# B&R Automation Studio project Y4_V3_1 (part 7)

#### Page13.st - Cyclic code
```iecst
(********************************************************************
 * COPYRIGHT --
 ********************************************************************
 * Program: Page13
 * File: Page13.st
 * Author: NickE
 * Created: January 31, 2013
 ********************************************************************
 * Implementation of program Page13
 ********************************************************************)

PROGRAM _CYCLIC

	//SETTINGS SCREEN
	Vis.P13.EnableIndex	:=	LIMIT(0,Vis.P13.EnableIndex,24)	;
	Vis.P13.Status[0]	:=	HIDE	;
	Vis.P13.Status[1]	:=	HIDE	;
	Vis.P13.Status[2]	:=	HIDE	;
	Vis.P13.Status[3]	:=	HIDE	;
	Vis.P13.Status[4]	:=	HIDE	;
	Vis.P13.Status[5]	:=	HIDE	;
	Vis.P13.Status[6]	:=	HIDE	;
	Vis.P13.Status[7]	:=	HIDE	;
	Vis.P13.Status[8]	:=	HIDE	;
	Vis.P13.Status[9]	:=	HIDE	;
	Vis.P13.Status[10]	:=	HIDE	;
	Vis.P13.Colour[1]	:=	BLUE	;
	Vis.P13.Colour[2]	:=	BLUE	;
	Vis.P13.Colour[3]	:=	BLUE	;
	Vis.P13.Colour[4]	:=	BLUE	;
	Vis.P13.Colour[5]	:=	BLUE	;
	Vis.P13.Colour[6]	:=	BLUE	;

	CASE Vis.P13.EnableIndex OF
		0:
			Vis.P13.Status[0]	:=	SHOW	;
			Vis.CalcBelt.Disp	:=	HIDE	;
		1:
			Vis.P13.Status[1]	:=	SHOW	;
			Vis.P13.Status[9]	:=	SHOW	;
			Vis.P13.Colour[1]	:=	BLUE_ACTIVE	;
		2:
			Vis.P13.Status[2]	:=	SHOW	;
			Vis.P13.Status[9]	:=	SHOW	;
			Vis.P13.Colour[2]	:=	BLUE_ACTIVE	;
			Vis.CalcBelt.Disp	:=	HIDE	;
		3:
			Vis.P13.Status[3]	:=	SHOW	;
			Vis.P13.Status[9]	:=	SHOW	;
			Vis.P13.Colour[3]	:=	BLUE_ACTIVE	;
			Vis.CalcBelt.Disp	:=	HIDE	;
		4:
			Vis.P13.Status[4]	:=	SHOW	;
			Vis.P13.Status[9]	:=	SHOW	;
			Vis.P13.Colour[4]	:=	BLUE_ACTIVE	;
			Vis.CalcBelt.Disp	:=	HIDE	;
		5:
			Vis.P13.Status[5]	:=	SHOW	;
			Vis.P13.Status[9]	:=	SHOW	;
			Vis.P13.Colour[5]	:=	BLUE_ACTIVE	;
			Vis.CalcBelt.Disp	:=	HIDE	;
		6:
			Vis.P13.Status[6]	:=	SHOW	;
			Vis.P13.Status[9]	:=	SHOW	;
			Vis.P13.Colour[6]	:=	BLUE_ACTIVE	;
			Vis.CalcBelt.Disp	:=	HIDE	;
		7:
			Vis.P13.Status[7]	:=	SHOW	;
			Vis.CalcBelt.Disp	:=	HIDE	;
		8:
			Vis.P13.Status[8]	:=	SHOW	;
			Vis.P13.Status[3]	:=	SHOW	;
			Vis.P13.Status[9]	:=	SHOW	;
			Vis.P13.Colour[3]	:=	BLUE_ACTIVE	;
			Vis.CalcBelt.Disp	:=	HIDE	;
		10:
			Vis.P13.Status[10]	:=	SHOW	;
			Vis.P13.Status[6]	:=	SHOW	;
			Vis.P13.Status[9]	:=	SHOW	;
			Vis.P13.Colour[6]	:=	BLUE_ACTIVE	;
			Vis.CalcBelt.Disp	:=	HIDE	;

	END_CASE

	//CALCULATE WHEN LAYER HAS CHANGED
	Vis.P13.Changed	:=	FALSE	;
	Vis.P13.New	:=	Vis.P13.EnableIndex	;
	IF(Vis.P13.New <> Vis.P13.Old) THEN
		Vis.P13.Changed	:=	TRUE	;
	END_IF
	IF EDGEPOS(Vis.P13.Changed) THEN
		Vis.P13Delays.EnableIndex	:=	24	;
		Vis.P13Servos.EnableIndex	:=	24	;
		Vis.P13System.EnableIndex	:=	24	;
		Vis.P13Timeouts.EnableIndex	:=	24	;
		Vis.P13Help1.EnableIndex	:=	24	;
		Vis.P13Help2.EnableIndex	:=	24	;
	END_IF
	Vis.P13.Old	:=	Vis.P13.EnableIndex	;

	//SETTINGS DELAYS SCREEN
	Vis.P13Delays.Status[0]	:=	HIDE	;
	Vis.P13Delays.Status[1]	:=	HIDE	;
	Vis.P13Delays.Status[2]	:=	HIDE	;
	Vis.P13Delays.Status[3]	:=	HIDE	;
	Vis.P13Delays.Status[4]	:=	HIDE	;
	Vis.P13Delays.Status[5]	:=	HIDE	;
	Vis.P13Delays.Status[6]	:=	HIDE	;
	Vis.P13Delays.Status[7]	:=	HIDE	;
	Vis.P13Delays.Status[8]	:=	HIDE	;
	Vis.P13Delays.Status[9]	:=	HIDE	;
	Vis.P13Delays.Status[10]	:=	HIDE	;
	Vis.P13Delays.Colour[0]	:=	BLUE	;
	Vis.P13Delays.Colour[1]	:=	BLUE	;
	Vis.P13Delays.Colour[2]	:=	BLUE	;
	Vis.P13Delays.Colour[3]	:=	BLUE	;
	Vis.P13Delays.Colour[4]	:=	BLUE	;
	Vis.P13Delays.Colour[5]	:=	BLUE	;
	Vis.P13Delays.Colour[6]	:=	BLUE	;
	Vis.P13Delays.Colour[7]	:=	BLUE	;
	Vis.P13Delays.Colour[8]	:=	BLUE	;

	CASE Vis.P13Delays.EnableIndex OF
		0..8://LayerDelay[1..9]
			Vis.P13Delays.Status[Vis.P13Delays.EnableIndex]	:=	SHOW	;
			Vis.P13Delays.Colour[Vis.P13Delays.EnableIndex]	:=	BLUE_ACTIVE	;
			Vis.P13Delays.Status[9]	:=	SHOW	;//LayerDelays
			Vis.P13.Status[1]	:=	HIDE	;//Layer2
			Vis.P13.Status[9]	:=	HIDE	;//Layers
		10:
			Vis.P13Delays.Status[10]	:=	SHOW	;
	END_CASE

	CASE Vis.P13Delays.EnableIndex OF
		0,3,4,7,8,24:
			Vis.CalcBelt.Disp	:=	HIDE	;
	END_CASE

	//CALCULATE WHEN LAYER HAS CHANGED
	Vis.P13Delays.Changed	:=	FALSE	;
	Vis.P13Delays.New	:=	Vis.P13Delays.EnableIndex	;
	IF(Vis.P13Delays.New <> Vis.P13Delays.Old) THEN
		Vis.P13Delays.Changed	:=	TRUE	;
	END_IF
	IF EDGEPOS(Vis.P13Delays.Changed) THEN
		Vis.P13Help1.EnableIndex	:=	24	;
		Vis.P13Help2.EnableIndex	:=	24	;
	END_IF
	Vis.P13Delays.Old	:=	Vis.P13Delays.EnableIndex	;

	//CALCULATOR FOR BELT DISPLAY
	IF (Vis.CalcBelt.Disp = SHOW) THEN
		IF (Vis.CalcBelt.Delay) THEN
			Vis.CalcBelt.Adjust	:= 	1 - ((Vis.CalcBelt.Unground + 300)/(Speeds.SpeedSeam/6))	;
		ELSE
			Vis.CalcBelt.Adjust	:= 	(Vis.CalcBelt.Unground + 300)/(Speeds.SpeedSeam/6);
		END_IF
		Vis.CalcBelt.New	:= 	(Vis.CalcBelt.Current + Vis.CalcBelt.Adjust)	;

		IF (Vis.CalcBelt.Unground = 0) THEN
			Vis.CalcBelt.Adjust	:= 	0	;
			Vis.CalcBelt.New	:= 	0	;
		END_IF
	END_IF

	//SETTINGS DRIVES SCREEN
	Vis.P13Drives.Status[0]	:=	HIDE	;
	Vis.P13Drives.Status[1]	:=	HIDE	;
	Vis.P13Drives.Status[2]	:=	HIDE	;
	Vis.P13Drives.Status[3]	:=	HIDE	;
	Vis.P13Drives.Status[4]	:=	HIDE	;
	Vis.P13Drives.Status[5]	:=	HIDE	;
	Vis.P13Drives.Status[6]	:=	HIDE	;
	Vis.P13Drives.Status[7]	:=	HIDE	;
	Vis.P13Drives.Status[8]	:=	HIDE	;
	Vis.P13Drives.Status[9]	:=	HIDE	;
	Vis.P13Drives.Status[10]:=	HIDE	;
	Vis.P13Drives.Status[11]:=	HIDE	;
	Vis.P13Drives.Status[12]:=	HIDE	;
	Vis.P13Drives.Status[13]:=	HIDE	;
	Vis.P13Drives.Status[14]:=	HIDE	;
	Vis.P13Drives.Status[15]:=	HIDE	;
	Vis.P13Drives.Status[20]:=	HIDE	;
	Vis.P13Drives.Status[21]:=	HIDE	;
	Vis.P13Drives.Status[22]:=	HIDE	;
	Vis.P13Drives.Colour[0]	:=	BLUE	;
	Vis.P13Drives.Colour[1]	:=	BLUE	;
	Vis.P13Drives.Colour[2]	:=	BLUE	;
	Vis.P13Drives.Colour[3]	:=	BLUE	;
	Vis.P13Drives.Colour[4]	:=	BLUE	;
	Vis.P13Drives.Colour[5]	:=	BLUE	;
	Vis.P13Drives.Colour[6]	:=	BLUE	;

	CASE Vis.P13Drives.EnableIndex OF
		0..6:
			Vis.P13Drives.Status[Vis.P13Drives.EnableIndex]	:=	SHOW	;
			Vis.P13Drives.Colour[Vis.P13Drives.EnableIndex]	:=	BLUE_ACTIVE	;
			Vis.P13Drives.Status[9]	:=	SHOW	;
			Vis.P13.Status[2]	:=	HIDE	;
			Vis.P13.Status[9]	:=	HIDE	;
			IF(Level.Level > SUPERVISOR) THEN
				Vis.P13Drives.Status[Vis.P13Drives.EnableIndex + 9]	:=	SHOW	;
			END_IF
		7:
			Vis.P13Drives.Status[7]	:=	SHOW	;
		8:
			Vis.P13Drives.Status[8]	:=	SHOW	;
	END_CASE

	CASE Vis.P13Drives.EnableIndex OF
		4:
			CASE InvPerms.CLB.Analog OF
				NO_ANALOG:
					AnalogStore.CLB.DisplayRaw := 0 ;
					AnalogStore.CLB.DisplaySpeed :=	0.0 ;
					AnalogStore.CLB.DisplayAnalog := 0.0 ;
				VOLTAGE_TYPE_1:
					AnalogStore.CLB.DisplayRaw := CLB.Input.AI1R ;
					AnalogStore.CLB.DisplaySpeed := AnalogPerm.CLB.V1.ActSpeed ;
					AnalogStore.CLB.DisplayAnalog := AnalogPerm.CLB.V1.ActAnalog ;
				CURRENT_TYPE_1:
					AnalogStore.CLB.DisplayRaw := CLB.Input.AI3R ;
					AnalogStore.CLB.DisplaySpeed := AnalogPerm.CLB.C1.ActSpeed ;
					AnalogStore.CLB.DisplayAnalog := AnalogPerm.CLB.C1.ActAnalog ;
				CURRENT_TYPE_2:
					AnalogStore.CLB.DisplayRaw := CLB.Input.AI3R ;
					AnalogStore.CLB.DisplaySpeed := AnalogPerm.CLB.C2.ActSpeed ;
					AnalogStore.CLB.DisplayAnalog := AnalogPerm.CLB.C2.ActAnalog ;
			END_CASE

			IF(AnalogStore.CLB.RecordStart) THEN
				Vis.P13Drives.Status[22]	:=	SHOW	;
			END_IF
			IF(AnalogStore.CLB.RecordConfirm) THEN
				CASE InvPerms.CLB.Analog OF
					VOLTAGE_TYPE_1:
						AnalogStore.CLB.DisplayRaw	:=	CLB.Input.AI1R	;
						AnalogPerm.CLB.V1.ActAnalog	:=	UINT_TO_REAL(AnalogStore.CLB.DisplayRaw)	;
						AnalogPerm.CLB.V1.ActSpeed	:=	AnalogStore.CLB.SpeedDisp	;
					CURRENT_TYPE_1:
						AnalogStore.CLB.DisplayRaw	:=	CLB.Input.AI3R	;
						AnalogPerm.CLB.C1.ActAnalog	:=	UINT_TO_REAL(AnalogStore.CLB.DisplayRaw)	;
						AnalogPerm.CLB.C1.ActSpeed	:=	AnalogStore.CLB.SpeedDisp	;
					CURRENT_TYPE_2:
						AnalogStore.CLB.DisplayRaw	:=	CLB.Input.AI3R	;
						AnalogPerm.CLB.C2.ActAnalog	:=	UINT_TO_REAL(AnalogStore.CLB.DisplayRaw)	;
						AnalogPerm.CLB.C2.ActSpeed	:=	AnalogStore.CLB.SpeedDisp	;
				END_CASE
				AnalogStore.CLB.RecordStart	:=	FALSE	;
				AnalogStore.CLB.RecordConfirm	:=	FALSE	;
			END_IF
		ELSE
			AnalogStore.CLB.RecordStart	:=	FALSE	;
			AnalogStore.CLB.RecordConfirm	:=	FALSE	;
	END_CASE

	//CALCULATE WHEN LAYER HAS CHANGED
	Vis.P13Drives.Changed	:=	FALSE	;
	Vis.P13Drives.New	:=	Vis.P13Drives.EnableIndex	;
	IF(Vis.P13Drives.New <> Vis.P13Drives.Old) THEN
		Vis.P13Drives.Changed	:=	TRUE	;
	END_IF
	IF EDGEPOS(Vis.P13Drives.Changed) THEN
		Vis.P13Help1.EnableIndex	:=	24	;
		Vis.P13Help2.EnableIndex	:=	24	;
	END_IF
	Vis.P13Drives.Old	:=	Vis.P13Drives.EnableIndex	;

	//SETTINGS SERVOS SCREEN
	Vis.P13Servos.Status[0]	:=	HIDE	;
	Vis.P13Servos.Status[1]	:=	HIDE	;
	Vis.P13Servos.Status[2]	:=	HIDE	;
	Vis.P13Servos.Status[3]	:=	HIDE	;
	Vis.P13Servos.Status[4]	:=	HIDE	;
	Vis.P13Servos.Status[5]	:=	HIDE	;
	Vis.P13Servos.Status[6]	:=	HIDE	;
	Vis.P13Servos.Status[7]	:=	HIDE	;
	Vis.P13Servos.Status[8]	:=	HIDE	;
	Vis.P13Servos.Status[9]	:=	HIDE	;
	Vis.P13Servos.Colour[0]	:=	BLUE	;
	Vis.P13Servos.Colour[1]	:=	BLUE	;
	Vis.P13Servos.Colour[2]	:=	BLUE	;
	Vis.P13Servos.Colour[3]	:=	BLUE	;
	Vis.P13Servos.Colour[4]	:=	BLUE	;
	Vis.P13Servos.Colour[5]	:=	BLUE	;
	Vis.P13Servos.Colour[6]	:=	BLUE	;

	CASE Vis.P13Servos.EnableIndex OF
		0..6:
			Vis.P13Servos.Status[Vis.P13Servos.EnableIndex]	:=	SHOW	;
			Vis.P13Servos.Colour[Vis.P13Servos.EnableIndex]	:=	BLUE_ACTIVE	;
			Vis.P13Servos.Status[9]	:=	SHOW	;
			Vis.P13.Status[2]	:=	HIDE	;
			Vis.P13.Status[9]	:=	HIDE	;
		7:
			Vis.P13Servos.Status[7]	:=	SHOW	;
		8:
			Vis.P13Servos.Status[8]	:=	SHOW	;
	END_CASE

	//CALCULATE WHEN LAYER HAS CHANGED
	Vis.P13Servos.Changed	:=	FALSE	;
	Vis.P13Servos.New	:=	Vis.P13Servos.EnableIndex	;
	IF(Vis.P13Servos.New <> Vis.P13Servos.Old) THEN
		Vis.P13Servos.Changed	:=	TRUE	;
	END_IF
	IF EDGEPOS(Vis.P13Servos.Changed) THEN
		Vis.P13Help1.EnableIndex	:=	24	;
		Vis.P13Help2.EnableIndex	:=	24	;
	END_IF
	Vis.P13Servos.Old	:=	Vis.P13Servos.EnableIndex	;

	//SETTINGS SYSTEM SCREEN
	Vis.P13System.Status[0]	:=	HIDE	;
	Vis.P13System.Status[1]	:=	HIDE	;
	Vis.P13System.Status[2]	:=	HIDE	;
	Vis.P13System.Status[3]	:=	HIDE	;
	Vis.P13System.Status[4]	:=	HIDE	;
	Vis.P13System.Status[5]	:=	HIDE	;
	Vis.P13System.Status[6]	:=	HIDE	;
	Vis.P13System.Status[7]	:=	HIDE	;
	Vis.P13System.Status[8]	:=	HIDE	;
	Vis.P13System.Status[9]	:=	HIDE	;
	Vis.P13System.Colour[0]	:=	BLUE	;
	Vis.P13System.Colour[1]	:=	BLUE	;
	Vis.P13System.Colour[2]	:=	BLUE	;
	Vis.P13System.Colour[3]	:=	BLUE	;
	Vis.P13System.Colour[4]	:=	BLUE	;
	Vis.P13System.Colour[5]	:=	BLUE	;
	Vis.P13System.Colour[6]	:=	BLUE	;

	CASE Vis.P13System.EnableIndex OF
		0..6:
			Vis.P13System.Status[Vis.P13System.EnableIndex]	:=	SHOW	;
			Vis.P13System.Colour[Vis.P13System.EnableIndex]	:=	BLUE_ACTIVE	;
			Vis.P13System.Status[9]	:=	SHOW	;
			Vis.P13.Status[4]	:=	HIDE	;
			Vis.P13.Status[9]	:=	HIDE	;
		7:
			Vis.P13System.Status[7]	:=	SHOW	;
		8:
			Vis.P13System.Status[8]	:=	SHOW	;
	END_CASE

	//CALCULATE WHEN LAYER HAS CHANGED
	Vis.P13System.Changed	:=	FALSE	;
	Vis.P13System.New	:=	Vis.P13System.EnableIndex	;
	IF(Vis.P13System.New <> Vis.P13System.Old) THEN
		Vis.P13System.Changed	:=	TRUE	;
	END_IF
	IF EDGEPOS(Vis.P13System.Changed) THEN
		Vis.P13Help1.EnableIndex	:=	24	;
		Vis.P13Help2.EnableIndex	:=	24	;
	END_IF
	Vis.P13System.Old	:=	Vis.P13System.EnableIndex	;

	//SETTINGS TIMEOUT SCREEN
	Vis.P13Timeouts.Status[0]	:=	HIDE	;
	Vis.P13Timeouts.Status[1]	:=	HIDE	;
	Vis.P13Timeouts.Status[2]	:=	HIDE	;
	Vis.P13Timeouts.Status[3]	:=	HIDE	;
	Vis.P13Timeouts.Status[4]	:=	HIDE	;
	Vis.P13Timeouts.Status[5]	:=	HIDE	;
	Vis.P13Timeouts.Status[6]	:=	HIDE	;
	Vis.P13Timeouts.Status[7]	:=	HIDE	;
	Vis.P13Timeouts.Status[8]	:=	HIDE	;
	Vis.P13Timeouts.Status[9]	:=	HIDE	;
	Vis.P13Timeouts.Colour[0]	:=	BLUE	;
	Vis.P13Timeouts.Colour[1]	:=	BLUE	;
	Vis.P13Timeouts.Colour[2]	:=	BLUE	;
	Vis.P13Timeouts.Colour[3]	:=	BLUE	;
	Vis.P13Timeouts.Colour[4]	:=	BLUE	;
	Vis.P13Timeouts.Colour[5]	:=	BLUE	;
	Vis.P13Timeouts.Colour[6]	:=	BLUE	;

	CASE Vis.P13Timeouts.EnableIndex OF
		0..6:
			Vis.P13Timeouts.Status[Vis.P13Timeouts.EnableIndex]	:=	SHOW	;
			Vis.P13Timeouts.Colour[Vis.P13Timeouts.EnableIndex]	:=	BLUE_ACTIVE	;
			Vis.P13Timeouts.Status[9]	:=	SHOW	;
			Vis.P13.Status[5]	:=	HIDE	;
			Vis.P13.Status[9]	:=	HIDE	;
		7:
			Vis.P13Timeouts.Status[7]	:=	SHOW	;
		8:
			Vis.P13Timeouts.Status[8]	:=	SHOW	;
	END_CASE

	//CALCULATE WHEN LAYER HAS CHANGED
	Vis.P13Timeouts.Changed	:=	FALSE	;
	Vis.P13Timeouts.New	:=	Vis.P13Timeouts.EnableIndex	;
	IF(Vis.P13Timeouts.New <> Vis.P13Timeouts.Old) THEN
		Vis.P13Timeouts.Changed	:=	TRUE	;
	END_IF
	IF EDGEPOS(Vis.P13Timeouts.Changed) THEN
		Vis.P13Help1.EnableIndex	:=	24	;
		Vis.P13Help2.EnableIndex	:=	24	;
	END_IF
	Vis.P13Timeouts.Old	:=	Vis.P13Timeouts.EnableIndex	;

	//HELP LAYERS CONTROL
	memcpy(ADR(Vis.P13Help1.Status),ADR(Vis.HideAll),SIZEOF(Vis.HideAll));
	Vis.P13Help1.Colour[0]	:=	BLUE	;
	Vis.P13Help1.Colour[1]	:=	BLUE	;
	Vis.P13Help1.Colour[2]	:=	BLUE	;
	Vis.P13Help1.Colour[3]	:=	BLUE	;
	Vis.P13Help1.Colour[4]	:=	BLUE	;
	Vis.P13Help1.Colour[5]	:=	BLUE	;
	Vis.P13Help1.Colour[6]	:=	BLUE	;
	Vis.P13Help1.Colour[7]	:=	BLUE	;
	Vis.P13Help1.Colour[8]	:=	BLUE	;
	Vis.P13Help1.Colour[9]	:=	BLUE	;

	CASE Vis.P13Help1.EnableIndex OF
		0..23:
			Vis.P13Help1.Status[Vis.P13Help1.EnableIndex]	:=	SHOW	;
		24:
			Vis.P13Help1.Index	:=	0	;
	END_CASE

	CASE Vis.P13Help1.Index OF
		0..9:
			Vis.P13Help1.Colour[Vis.P13Help1.Index]	:=	BLUE_ACTIVE	;
	END_CASE

	//HELP LAYERS CONTROL 2
	memcpy(ADR(Vis.P13Help2.Status),ADR(Vis.HideAll),SIZEOF(Vis.HideAll));
	Vis.P13Help2.Colour[0]	:=	BLUE	;
	Vis.P13Help2.Colour[1]	:=	BLUE	;
	Vis.P13Help2.Colour[2]	:=	BLUE	;
	Vis.P13Help2.Colour[3]	:=	BLUE	;
	Vis.P13Help2.Colour[4]	:=	BLUE	;
	Vis.P13Help2.Colour[5]	:=	BLUE	;
	Vis.P13Help2.Colour[6]	:=	BLUE	;
	Vis.P13Help2.Colour[7]	:=	BLUE	;
	Vis.P13Help2.Colour[8]	:=	BLUE	;
	Vis.P13Help2.Colour[9]	:=	BLUE	;
	Vis.P13Help2.Colour[10]	:=	BLUE	;

	CASE Vis.P13Help2.EnableIndex OF
		0..23:
			Vis.P13Help2.Status[Vis.P13Help2.EnableIndex]	:=	SHOW	;
		24:
			Vis.P13Help2.Index	:=	0	;
	END_CASE

	CASE Vis.P13Help2.Index OF
		0..10:
			Vis.P13Help2.Colour[Vis.P13Help2.Index]	:=	BLUE_ACTIVE	;
	END_CASE

END_PROGRAM
```

### Program Logical/VisControl/HMIControl/Page14 (IEC) - Drives screen

#### Page14.st - Cyclic code
```iecst
(********************************************************************
 * COPYRIGHT --
 ********************************************************************
 * Program: Page14
 * File: Page14.st
 * Author: NickE
 * Created: January 31, 2013
 ********************************************************************
 * Implementation of program Page14
 ********************************************************************)

PROGRAM _CYCLIC

	//DRIVES SCREEN
	memcpy(ADR(Vis.P14.Status),ADR(Vis.HideAll),SIZEOF(Vis.HideAll));
	Vis.P14.Colour[0]	:=	VIOLET	;
	Vis.P14.Colour[1]	:=	VIOLET	;
	Vis.P14.Colour[2]	:=	VIOLET	;
	Vis.P14.Colour[3]	:=	VIOLET	;
	Vis.P14.Colour[4]	:=	VIOLET	;
	Vis.P14.Colour[5]	:=	VIOLET	;
	Vis.P14.Colour[6]	:=	VIOLET	;

	CASE Vis.P14.EnableIndex OF
		0..6:
			Vis.P14.Status[Vis.P14.EnableIndex]	:=	SHOW	;
			Vis.P14.Colour[Vis.P14.EnableIndex]	:=	VIOLET_ACTIVE	;
	END_CASE

	IF (Control.Test) THEN
		Vis.P14.Status[8]	:=	SHOW	;
	END_IF

	IF(Control.Test) THEN
		Vis.P14.Status[9]	:=	SHOW	;
	END_IF

	//CALCULATE WHEN LAYER HAS CHANGED
	Vis.P14.Changed	:=	FALSE	;
	Vis.P14.New	:=	Vis.P14.EnableIndex	;
	IF(Vis.P14.New <> Vis.P14.Old) THEN
		Vis.P14.Changed	:=	TRUE	;
	END_IF
	IF EDGEPOS(Vis.P14.Changed) THEN
		Vis.P14Layer.EnableIndex	:=	24	;
		Vis.P14Status.EnableIndex	:=	24	;
		Vis.P14Help.EnableIndex		:=	24	;
		//		Vis.CalcFreq.Disp				:=	HIDE	;
	END_IF
	Vis.P14.Old	:=	Vis.P14.EnableIndex	;

	memcpy(ADR(Vis.P14Layer.Status),ADR(Vis.HideAll),SIZEOF(Vis.HideAll));

	CASE Vis.P14Layer.EnableIndex OF
		0..19:
			Vis.P14Layer.Status[Vis.P14Layer.EnableIndex]	:=	SHOW	;
//		24:
//			Vis.CalcFreq.Disp	:=	HIDE	;
	END_CASE

	IF NOT(Control.Test) THEN
		Vis.P14Layer.EnableIndex	:= 24	;
	END_IF

	memcpy(ADR(Vis.P14Status.Status),ADR(Vis.HideAll),SIZEOF(Vis.HideAll));

	CASE Vis.P14Status.EnableIndex OF
		0..19:
			Vis.P14Status.Status[Vis.P14Status.EnableIndex]	:=	SHOW	;
	END_CASE

	memcpy(ADR(Vis.P14Help.Status),ADR(Vis.HideAll),SIZEOF(Vis.HideAll));

	CASE Vis.P14Help.EnableIndex OF
		0..15:
			Vis.P14Help.Status[Vis.P14Help.EnableIndex]	:=	SHOW	;
	END_CASE

	//DISPLAY INVERTER RESET BUTTON
	FOR i := 16 TO 31 DO
		IF(SysTemp.Alarms[i])THEN
			Vis.P14.Status[23]	:=	SHOW	;
		END_IF
	END_FOR
	IF(InvReset.Auto) AND(CL1.Input.Fault) THEN
		CL1.Output.CMDD_07	:=	TRUE	;
	END_IF
	IF(InvReset.Auto) AND(CS1.Input.Fault) THEN
		CS1.Output.CMDD_07	:=	TRUE	;
	END_IF
	IF(InvReset.Auto) AND(CV1.Input.Fault) THEN
		CV1.Output.CMDD_07	:=	TRUE	;
	END_IF
	IF(InvReset.Auto) AND(CC1.Input.Fault) THEN
		CC1.Output.CMDD_07	:=	TRUE	;
	END_IF
	IF(InvReset.Auto) AND(CC2.Input.Fault) THEN
		CC2.Output.CMDD_07	:=	TRUE	;
	END_IF
	IF(InvReset.Auto) AND(CS2.Input.Fault) THEN
		CS2.Output.CMDD_07	:=	TRUE	;
	END_IF
	IF(InvReset.Auto) AND(CV2.Input.Fault) THEN
		CV2.Output.CMDD_07	:=	TRUE	;
	END_IF
	IF(InvReset.Auto) AND(CC3.Input.Fault) THEN
		CC3.Output.CMDD_07	:=	TRUE	;
	END_IF
	IF(InvReset.Auto) AND(CC4.Input.Fault) THEN
		CC4.Output.CMDD_07	:=	TRUE	;
	END_IF
	IF(InvReset.Auto) AND(CB1.Input.Fault) THEN
		CB1.Output.CMDD_07	:=	TRUE	;
	END_IF
	IF(InvReset.Auto) AND(CB2.Input.Fault) THEN
		CB2.Output.CMDD_07	:=	TRUE	;
	END_IF
	IF(InvReset.Auto) AND(CRB.Input.Fault) THEN
		CRB.Output.CMDD_07	:=	TRUE	;
	END_IF
	IF(InvReset.Auto) AND(CRE.Input.Fault) THEN
		CRE.Output.CMDD_07	:=	TRUE	;
	END_IF
	IF(InvReset.Auto) AND(CLB.Input.Fault) THEN
		CLB.Output.CMDD_07	:=	TRUE	;
	END_IF

END_PROGRAM
```

### Program Logical/VisControl/HMIControl/Page15 (IEC) - Servo screen controls

#### Page15.st - Cyclic code
```iecst
(********************************************************************
 * COPYRIGHT --
 ********************************************************************
 * Program: Page15
 * File: Page15.st
 * Author: nicke
 * Created: February 04, 2013
 ********************************************************************
 * Implementation of program Page15
 ********************************************************************)

PROGRAM _CYCLIC

	//SERVOS SCREEN
	memcpy(ADR(Vis.P15.Status),ADR(Vis.HideAll),SIZEOF(Vis.HideAll));
	Vis.P15.Colour[0]	:=	GREEN1	;
	Vis.P15.Colour[1]	:=	GREEN1	;
	Vis.P15.Colour[2]	:=	GREEN1	;
	Vis.P15.Colour[3]	:=	GREEN1	;
	Vis.P15.Colour[4]	:=	GREEN1	;
	Vis.P15.Colour[5]	:=	GREEN1	;
	Vis.P15.Colour[6]	:=	GREEN1	;

	CASE Vis.P15.EnableIndex OF
		0..6:
			Vis.P15.Status[Vis.P15.EnableIndex]	:=	SHOW	;
			Vis.P15.Colour[Vis.P15.EnableIndex]	:=	GREEN1_ACTIVE	;
	END_CASE

	IF(Control.Test) THEN
		Vis.P15.Status[8]	:=	SHOW	;
		//	ELSE
		//		Vis.P15Layer.EnableIndex	:=	24	;
	END_IF

	//CALCULATE WHEN LAYER HAS CHANGED
	Vis.P15.Changed	:=	FALSE	;
	Vis.P15.New	:=	Vis.P15.EnableIndex	;
	IF(Vis.P15.New <> Vis.P15.Old) THEN
		Vis.P15.Changed	:=	TRUE	;
	END_IF
	IF EDGEPOS(Vis.P15.Changed) THEN
		Vis.P15Layer.EnableIndex	:=	24	;
	END_IF
	Vis.P15.Old	:=	Vis.P15.EnableIndex	;

	memcpy(ADR(Vis.P15Layer.Status),ADR(Vis.HideAll),SIZEOF(Vis.HideAll));

	CASE Vis.P15Layer.EnableIndex OF
		0..15:
			Vis.P15Layer.Status[Vis.P15Layer.EnableIndex]	:=	SHOW	;
	END_CASE

	IF(Control.Test) THEN
		TestServos	:=	TRUE	;
	ELSE
		TestServos	:=	FALSE	;
		Vis.P15Layer.Status[0]	:=	HIDE	;
		Vis.P15Layer.Status[1]	:=	HIDE	;
		Vis.P15Layer.Status[2]	:=	HIDE	;
	END_IF

	Ax1.Seek2Runtime	:=	(BOOL_TO_USINT(Ax1.Block));
	Ax2.Seek2Runtime	:=	(BOOL_TO_USINT(Ax2.Block));

END_PROGRAM
```

### Program Logical/VisControl/HMIControl/Page16 (IEC) - Remote screen control

#### Page16.st - Cyclic code
```iecst
(********************************************************************
 * COPYRIGHT --
 ********************************************************************
 * Program: Page16
 * File: Page16.st
 * Author: nicke
 * Created: February 07, 2013
 ********************************************************************
 * Implementation of program Page16
 ********************************************************************)

PROGRAM _CYCLIC

	//REMOTE SCREEN
	memcpy(ADR(Vis.P16.Status),ADR(Vis.HideAll),SIZEOF(Vis.HideAll));
	Vis.P16.Colour[0]	:=	LIGHTBLUE	;
	Vis.P16.Colour[1]	:=	LIGHTBLUE	;
	Vis.P16.Colour[2]	:=	LIGHTBLUE	;
	Vis.P16.Colour[3]	:=	LIGHTBLUE	;
	Vis.P16.Colour[4]	:=	LIGHTBLUE	;
	Vis.P16.Colour[5]	:=	LIGHTBLUE	;
	Vis.P16.Colour[6]	:=	LIGHTBLUE	;
	Vis.P16.Colour[7]	:=	LIGHTBLUE	;
	Vis.P16.Colour[8]	:=	LIGHTBLUE	;
	Vis.P16.Colour[9]	:=	LIGHTBLUE	;
	Vis.P16.Colour[10]	:=	LIGHTBLUE	;

	CASE Vis.P16.EnableIndex OF
		0..7,9,10:
			Vis.P16.Status[Vis.P16.EnableIndex]	:=	SHOW	;
			Vis.P16.Colour[Vis.P16.EnableIndex]	:=	LIGHTBLUE_ACTIVE	;
	END_CASE

	IF(Control.Test) THEN
		Vis.P16.Status[8]	:=	SHOW	;
	ELSE
		Vis.P16.EnableIndex	:= LIMIT(0, Vis.P16.EnableIndex, 5);//ALTER Limit max dependent on number of IO screens, 5=6 screens ETC...
	END_IF

	//CALCULATE WHEN LAYER HAS CHANGED
	Vis.P16.Changed	:=	FALSE	;
	Vis.P16.New	:=	Vis.P16.EnableIndex	;
	IF(Vis.P16.New <> Vis.P16.Old) THEN
		Vis.P16.Changed	:=	TRUE	;
	END_IF
	IF EDGEPOS(Vis.P16.Changed) THEN
		Vis.P16Layer.EnableIndex	:=	24	;
	END_IF
	Vis.P16.Old	:=	Vis.P16.EnableIndex	;

	memcpy(ADR(Vis.P16Layer.Status),ADR(Vis.HideAll),SIZEOF(Vis.HideAll));

	CASE Vis.P16Layer.EnableIndex OF
		0..15:
			Vis.P16Layer.Status[Vis.P16Layer.EnableIndex]	:=	SHOW	;
	END_CASE

	//Declaration to enable use of variables on screen
	X2XModule	;

END_PROGRAM
```

### Program Logical/VisControl/HMIControl/Page17 (IEC) - Alarm screen control

#### Page17.st - Cyclic code
```iecst
(********************************************************************
 * COPYRIGHT -ASHTON INDUSTRIAL 2016-
 ********************************************************************
 * Program: Page17
 * File: Page17.st
 * Author: NE
 ********************************************************************)

PROGRAM _CYCLIC

	Alarm.Control := 3 ;  	//Enable Alarm Index selection
	Alarm.Group := 1 ;	// Equals alarm group index
	Alarm.Alarm := 0 ;	// Not used
	Alarm.Priority := 0 ;	// Not used

	// Convert alarm inputs to alarm array
	SysTemp.Alarms[0] := MS1Belt1.Trip ;
	SysTemp.Alarms[1] := MS2Belt2.Trip ;
	SysTemp.Alarms[2] := MS3Belt3.Trip ;
	SysTemp.Alarms[3] := MS4Belt4.Trip ;
	SysTemp.Alarms[4] := MS5Belt5.Trip ;
	SysTemp.Alarms[5] := MS6Belt6.Trip ;
	SysTemp.Alarms[6] := MS7Belt7.Trip ;
	SysTemp.Alarms[7] := MS8Belt8.Trip ;
	SysTemp.Alarms[8] := MS9Vac1.Trip ;
	SysTemp.Alarms[9] := MS10Vac2.Trip ;
	SysTemp.Alarms[10] := MS11Vac3.Trip ;
	SysTemp.Alarms[11] := MS12Vac4.Trip ;
	SysTemp.Alarms[12] := MS13Water1.Trip ;
	SysTemp.Alarms[13] := MS14Water2.Trip ;
	SysTemp.Alarms[14] := (CL1.Input.Fault) ;
	SysTemp.Alarms[15] := (CS1.Input.Fault) ;
	SysTemp.Alarms[16] := (CV1.Input.Fault) ;
	SysTemp.Alarms[17] := (CC1.Input.Fault) ;
	SysTemp.Alarms[18] := (CC2.Input.Fault) ;
	SysTemp.Alarms[19] := (CS2.Input.Fault) ;
	SysTemp.Alarms[20] := (CV2.Input.Fault) ;
	SysTemp.Alarms[21] := (CC3.Input.Fault) ;
	SysTemp.Alarms[22] := (CC4.Input.Fault) ;
	SysTemp.Alarms[23] := (CB1.Input.Fault) ;
	SysTemp.Alarms[24] := (CB2.Input.Fault) ;
	SysTemp.Alarms[25] := (CRB.Input.Fault) ;
	SysTemp.Alarms[26] := (CRE.Input.Fault) ;
	SysTemp.Alarms[27] := (CLB.Input.Fault) ;
	SysTemp.Alarms[28] ;
	SysTemp.Alarms[29] ;
	SysTemp.Alarms[30] ;
	SysTemp.Alarms[31] ;
	SysTemp.Alarms[32] ;
	SysTemp.Alarms[33] ;
	SysTemp.Alarms[39] := Ax1.Error AND(Control.Achieved1) ;
	SysTemp.Alarms[40] := Ax2.Error AND(Control.Achieved1) ;
	SysTemp.Alarms[41] := NOT(Servo1POT.In) ;
	SysTemp.Alarms[42] := NOT(Servo1NOT.In) ;
	SysTemp.Alarms[43] := NOT(Servo2POT.In) ;
	SysTemp.Alarms[44] := NOT(Servo2NOT.In) ;
	SysTemp.Alarms[50] := (X2XModule[5].Fuse) ;
	SysTemp.Alarms[51] := (X2XModule[6].Fuse) ;
	SysTemp.Alarms[52] := (X2XModule[7].Fuse) ;

	SysTemp.Alarm := FALSE ;
	FOR i := 0 TO 80 DO
		IF(SysTemp.Alarms[i]) THEN
			SysTemp.Alarm := TRUE ;
			EXIT ;
		END_IF
	END_FOR

END_PROGRAM
```

### Program Logical/VisControl/HMIControl/Page18 (IEC) - Warning screen control

#### Page18.st - Cyclic code
```iecst
(********************************************************************
 * COPYRIGHT --
 ********************************************************************
 * Program: Page18
 * File: Page18.st
 * Author: nicke
 * Created: April 30, 2013
 ********************************************************************
 * Implementation of program Page18
 ********************************************************************)

PROGRAM _CYCLIC

(* Section to control pop up warnings for flip arms *)
(*Seamer 1 Down *)
	Vis.FlipDisp1.Runtime1	:=	HIDE	;
	Vis.FlipDisp1.Runtime2	:=	HIDE	;
	Vis.FlipDisp1.Runtime3	:=	HIDE	;
	Vis.FlipDisp1.Runtime4	:=	HIDE	;

	IF ((Ax1.Active) OR NOT(Ax1.OriginSet)) AND NOT(Ax1.Block) AND(Control.Achieved1) THEN
		Vis.FlipDisp1.Runtime1	:=	SHOW	;
		Vis.FlipDisp1.TextIndex1	:=	BOOL_TO_USINT(NOT(S100Reed.In))	;
		Vis.FlipDisp1.TextIndex2	:=	BOOL_TO_USINT(NOT(S102Reed.In))	;
		Vis.FlipDisp1.TextIndex3	:=	BOOL_TO_USINT(NOT(S104Reed.In))	;
		Vis.FlipDisp1.TextIndex4	:=	BOOL_TO_USINT(NOT(S106Reed.In))	;
		Vis.FlipDisp1.TextIndex5	:=	BOOL_TO_USINT(NOT(S108Reed.In))	;
		Vis.FlipDisp1.TextIndex6	:=	BOOL_TO_USINT(NOT(S110Reed.In))	;
		Vis.FlipDisp1.TextIndex7	:=	BOOL_TO_USINT(NOT(S112Reed.In))	;
		Vis.FlipDisp1.TextIndex8	:=	BOOL_TO_USINT(NOT(S114Reed.In))	;
		Vis.FlipDisp1.TextIndex9	:=	BOOL_TO_USINT(NOT(S116Reed.In))	;
		Vis.FlipDisp1.TextIndex10	:=	BOOL_TO_USINT(NOT(S118Reed.In))	;
		CASE Perms.FLIPARMS1 OF
			3:
				Vis.FlipDisp1.Runtime2		:=	SHOW	;
			4:
				Vis.FlipDisp1.Runtime2		:=	SHOW	;
				Vis.FlipDisp1.Runtime3		:=	SHOW	;
			5:
				Vis.FlipDisp1.Runtime2		:=	SHOW	;
				Vis.FlipDisp1.Runtime3		:=	SHOW	;
				Vis.FlipDisp1.Runtime4		:=	SHOW	;
		END_CASE
	END_IF

	(* Seamer 1 Up *)
	Vis.FlipDisp1.Runtime5	:= HIDE	;
	Vis.FlipDisp1.Runtime6	:= HIDE	;
	Vis.FlipDisp1.Runtime7	:= HIDE	;
	Vis.FlipDisp1.Runtime8	:= HIDE	;
	Vis.FlipDisp1.Runtime9	:= HIDE	;
	Vis.FlipDisp1.TextIndex11	:=	BOOL_TO_USINT(NOT(S101Reed.In))	;
	Vis.FlipDisp1.TextIndex12	:=	BOOL_TO_USINT(NOT(S103Reed.In))	;
	Vis.FlipDisp1.TextIndex13	:=	BOOL_TO_USINT(NOT(S105Reed.In))	;
	Vis.FlipDisp1.TextIndex14	:=	BOOL_TO_USINT(NOT(S107Reed.In))	;
	Vis.FlipDisp1.TextIndex15	:=	BOOL_TO_USINT(NOT(S109Reed.In))	;
	Vis.FlipDisp1.TextIndex16	:=	BOOL_TO_USINT(NOT(S111Reed.In))	;
	Vis.FlipDisp1.TextIndex17	:=	BOOL_TO_USINT(NOT(S113Reed.In))	;
	Vis.FlipDisp1.TextIndex18	:=	BOOL_TO_USINT(NOT(S115Reed.In))	;
	Vis.FlipDisp1.TextIndex19	:=	BOOL_TO_USINT(NOT(S117Reed.In))	;
	Vis.FlipDisp1.TextIndex20	:=	BOOL_TO_USINT(NOT(S119Reed.In))	;
	CASE ArmsTemp1.CheckRaised OF
		0:	(* No arms up *)
		1:	(* 1 arm up *)
			Vis.FlipDisp1.Runtime5	:= SHOW	;
		2:	(* 2 arms up *)
			Vis.FlipDisp1.Runtime5	:= SHOW	;
			Vis.FlipDisp1.Runtime6	:= SHOW	;
		3:  (* 3 arms up *)
			Vis.FlipDisp1.Runtime5	:= SHOW	;
			Vis.FlipDisp1.Runtime6	:= SHOW	;
			Vis.FlipDisp1.Runtime7	:= SHOW	;
		4:	(* 4 arms up *)
			Vis.FlipDisp1.Runtime5	:= SHOW	;
			Vis.FlipDisp1.Runtime6	:= SHOW	;
			Vis.FlipDisp1.Runtime7	:= SHOW	;
			Vis.FlipDisp1.Runtime8	:= SHOW	;
		5:	(* 5 arms up *)
			Vis.FlipDisp1.Runtime5	:= SHOW	;
			Vis.FlipDisp1.Runtime6	:= SHOW	;
			Vis.FlipDisp1.Runtime7	:= SHOW	;
			Vis.FlipDisp1.Runtime8	:= SHOW	;
			Vis.FlipDisp1.Runtime9	:= SHOW	;
	END_CASE

	(* Seamer 2 Down *)
	Vis.FlipDisp2.Runtime1	:=	HIDE	;
	Vis.FlipDisp2.Runtime2	:=	HIDE	;
	Vis.FlipDisp2.Runtime3	:=	HIDE	;
	Vis.FlipDisp2.Runtime4	:=	HIDE	;

	IF ((Ax2.Active) OR NOT(Ax2.OriginSet)) AND NOT(Ax2.Block) AND(Control.Achieved1) THEN
		Vis.FlipDisp2.Runtime1	:=	SHOW	;
		Vis.FlipDisp2.TextIndex1	:=	BOOL_TO_USINT(NOT(S120Reed.In))	;
		Vis.FlipDisp2.TextIndex2	:=	BOOL_TO_USINT(NOT(S122Reed.In))	;
		Vis.FlipDisp2.TextIndex3	:=	BOOL_TO_USINT(NOT(S124Reed.In))	;
		Vis.FlipDisp2.TextIndex4	:=	BOOL_TO_USINT(NOT(S126Reed.In))	;
		Vis.FlipDisp2.TextIndex5	:=	BOOL_TO_USINT(NOT(S128Reed.In))	;
		Vis.FlipDisp2.TextIndex6	:=	BOOL_TO_USINT(NOT(S130Reed.In))	;
		Vis.FlipDisp2.TextIndex7	:=	BOOL_TO_USINT(NOT(S132Reed.In))	;
		Vis.FlipDisp2.TextIndex8	:=	BOOL_TO_USINT(NOT(S134Reed.In))	;
		Vis.FlipDisp2.TextIndex9	:=	BOOL_TO_USINT(NOT(S136Reed.In))	;
		Vis.FlipDisp2.TextIndex10	:=	BOOL_TO_USINT(NOT(S138Reed.In))	;
		CASE Perms.FLIPARMS2 OF
			3:
				Vis.FlipDisp2.Runtime2	:=	SHOW	;
			4:
				Vis.FlipDisp2.Runtime2	:=	SHOW	;
				Vis.FlipDisp2.Runtime3	:=	SHOW	;
			5:
				Vis.FlipDisp2.Runtime2	:=	SHOW	;
				Vis.FlipDisp2.Runtime3	:=	SHOW	;
				Vis.FlipDisp2.Runtime4	:=	SHOW	;
		END_CASE
	END_IF

	(* Seamer 2 Up *)
	Vis.FlipDisp2.Runtime5	:= HIDE	;
	Vis.FlipDisp2.Runtime6	:= HIDE	;
	Vis.FlipDisp2.Runtime7	:= HIDE	;
	Vis.FlipDisp2.Runtime8	:= HIDE	;
	Vis.FlipDisp2.Runtime9	:= HIDE	;
	Vis.FlipDisp2.TextIndex11	:=	BOOL_TO_USINT(NOT(S121Reed.In))	;
	Vis.FlipDisp2.TextIndex12	:=	BOOL_TO_USINT(NOT(S123Reed.In))	;
	Vis.FlipDisp2.TextIndex13	:=	BOOL_TO_USINT(NOT(S125Reed.In))	;
	Vis.FlipDisp2.TextIndex14	:=	BOOL_TO_USINT(NOT(S127Reed.In))	;
	Vis.FlipDisp2.TextIndex15	:=	BOOL_TO_USINT(NOT(S129Reed.In))	;
	Vis.FlipDisp2.TextIndex16	:=	BOOL_TO_USINT(NOT(S131Reed.In))	;
	Vis.FlipDisp2.TextIndex17	:=	BOOL_TO_USINT(NOT(S133Reed.In))	;
	Vis.FlipDisp2.TextIndex18	:=	BOOL_TO_USINT(NOT(S135Reed.In))	;
	Vis.FlipDisp2.TextIndex19	:=	BOOL_TO_USINT(NOT(S137Reed.In))	;
	Vis.FlipDisp2.TextIndex20	:=	BOOL_TO_USINT(NOT(S139Reed.In))	;
	CASE ArmsTemp2.CheckRaised OF
		0:	(* No arms up *)
		1:	(* 1 arm up *)
			Vis.FlipDisp2.Runtime5	:= SHOW	;
			Vis.FlipDisp2.Runtime6	:= SHOW	;
		2:	(* 2 arms up *)
			Vis.FlipDisp2.Runtime5	:= SHOW	;
			Vis.FlipDisp2.Runtime6	:= SHOW	;
			Vis.FlipDisp2.Runtime7	:= SHOW	;
		3:  (* 3 arms up *)
			Vis.FlipDisp2.Runtime5	:= SHOW	;
			Vis.FlipDisp2.Runtime6	:= SHOW	;
			Vis.FlipDisp2.Runtime7	:= SHOW	;
			Vis.FlipDisp2.Runtime8	:= SHOW	;
		4:	(* 4 arms up *)
			Vis.FlipDisp2.Runtime5	:= SHOW	;
			Vis.FlipDisp2.Runtime6	:= SHOW	;
			Vis.FlipDisp2.Runtime7	:= SHOW	;
			Vis.FlipDisp2.Runtime8	:= SHOW	;
			Vis.FlipDisp2.Runtime9	:= SHOW	;
	END_CASE

	//FILTER TO SHOW WARNINGS
	Warning.Control := 3 ; 	//Enable Alarm Index selection *)
	Warning.Group := 3 ;
	Warning.Alarm := 0 ;
	Warning.Priority := 0 ;

	Warn.Timeout[0] := Track001.TimeoutOUT ;
	Warn.Timeout[1] := Track002.TimeoutOUT ;
	Warn.Timeout[2] := Track003.TimeoutOUT ;
	Warn.Timeout[3] := Track101.TimeoutOUT ;
	Warn.Timeout[4] := Track102.TimeoutOUT ;
	Warn.Timeout[5] := Track104.TimeoutOUT ;
	Warn.Timeout[6] := Track106.TimeoutOUT ;
	Warn.Timeout[7] := Track111.TimeoutOUT ;
	Warn.Timeout[8] := Track112.TimeoutOUT ;
	Warn.Timeout[9] := Track113.TimeoutOUT ;
	Warn.Timeout[10] := Track201.TimeoutOUT ;
	Warn.Timeout[11] := Track202.TimeoutOUT ;
	Warn.Timeout[12] := Track204.TimeoutOUT ;
	Warn.Timeout[13] := Track207.TimeoutOUT ;
	Warn.Timeout[14] := Track301.TimeoutOUT ;
	Warn.Timeout[15] := Track401.TimeoutOUT ;
	Warn.Timeout[16] := Track412.TimeoutOUT ;
	Warn.Timeout[17] := Track413.TimeoutOUT ;
	Warn.Timeout[18] := Track414.TimeoutOUT ;
	Warn.Timeout[19] := Track503.TimeoutOUT ;
	Warn.Timeout[20] := Track504.TimeoutOUT ;
	Warn.Timeout[21] := Track506.TimeoutOUT ;
	Warn.Timeout[22] := Track602.TimeoutOUT ;
	Warn.Timeout[23] := Track801.TimeoutOUT ;
	Warn.Timeout[24] := Track803.TimeoutOUT ;
	Warn.Timeout[25] := Track804.TimeoutOUT ;
	Warn.Timeout[26] := Track805.TimeoutOUT ;
	Warn.Timeout[27] := Track811.TimeoutOUT ;
	Warn.Timeout[28] := Track821.TimeoutOUT ;
	Warn.Timeout[29] := Track512.TimeoutOUT ;

	FOR i:= 0 TO USINT_TO_INT(Warn.iMax) DO
		IF EDGEPOS(Warn.Timeout[i]) THEN
			Warn.Acks[i] := TRUE ;
		END_IF
	END_FOR

	FOR i:= 0 TO USINT_TO_INT(Warn.iMax) DO
		IF NOT(Warn.Timeout[i]) THEN
			Warn.Acks[i] := FALSE ;
		END_IF
	END_FOR

	//SET WARNING BIT ACTIVE WHEN TIMEOUT OCCURS
	FOR Warn.i:= 0 TO Warn.iMax DO
		IF Warn.Timeout[Warn.i] = TRUE THEN
			SysTemp.Warning :=  TRUE ;
			Warn.Button := SHOW ;
			EXIT;
		ELSE
			SysTemp.Warning := FALSE ;
			Warn.Button := HIDE ;
		END_IF
	END_FOR

	//Apply Warn.Block if EMO.Latch* are on
	IF EDGEPOS(EMO.Latch1) AND NOT(Warn.Block) THEN
		Warn.Block := TRUE ;
		Warn.BlockTemp := TRUE ;
	END_IF
	IF EDGEPOS(EMO.Latch2) AND NOT(Warn.Block) THEN
		Warn.Block := TRUE ;
		Warn.BlockTemp := TRUE ;
	END_IF

	IF EDGENEG(EMO.Latch1) AND NOT(EMO.Latch2) AND(Warn.BlockTemp) THEN
		Warn.Block := FALSE ;
		Warn.BlockTemp := FALSE ;
	END_IF
	IF EDGENEG(EMO.Latch2) AND NOT(EMO.Latch1) AND(Warn.BlockTemp) THEN
		Warn.Block := FALSE ;
		Warn.BlockTemp := FALSE ;
	END_IF

	//RESET ACK BITS IF TIMEOUT DISABLED
	IF(Warn.Block) THEN
		FOR Warn.Warningi:= 0 TO Warn.iMax DO
			Warn.Acks[Warn.Warningi]:= FALSE;
		END_FOR
	END_IF

	Warn.AckDisp	:= 	HIDE	;
	IF(SysTemp.Warning) THEN
		FOR Warn.Warningi:= 0 TO Warn.iMax DO
			IF (Warn.Acks[Warn.Warningi] = TRUE) THEN
				Warn.AckDisp	:= 	SHOW	;
				EXIT;
			ELSE
				Warn.AckDisp	:= 	HIDE	;
			END_IF
		END_FOR
	END_IF

	IF EDGEPOS(Warn.Ack) THEN
		Warn.Acks[Warn.Warningi]	:=	0	;
	END_IF

	//EVENTS
	SysTemp.Events[0] := Control.Start ;
	SysTemp.Events[1] := Control.Stop ;
	SysTemp.Events[2] := Control.EStop1 AND Control.Empty ;
	SysTemp.Events[3] := Control.EStop1 AND NOT Control.Empty ;
	SysTemp.Events[4] := SeamersII.Enable[1] ;
	SysTemp.Events[5] := SeamersII.Enable[2] ;
	SysTemp.Events[8] := SeamersII.AutoStart[0] ;
	SysTemp.Events[9] := SeamersII.AutoStart[1] ;
	SysTemp.Events[10] := SeamersII.AutoStart[2] ;
	SysTemp.Events[13] := Control.Achieved1 ;
	SysTemp.Events[14] := Control.Achieved2 ;
	SysTemp.Events[15] := Reset.Count ;
	SysTemp.Events[16] := Pause.Active ;

END_PROGRAM
```

### Program Logical/VisControl/HMIControl/Page20 (IEC) - Ashton tech screen control

#### Page20.st - Cyclic code
```iecst
(********************************************************************
 * COPYRIGHT --
 ********************************************************************
 * Program: P20
 * File: P20.st
 * Author: nicke
 * Created: February 08, 2013
 ********************************************************************
 * Implementation of program P20
 ********************************************************************)

PROGRAM _CYCLIC

	//ASHTON TECH SCREEN
	memcpy(ADR(Vis.P20.Status),ADR(Vis.HideAll),SIZEOF(Vis.HideAll));

	CASE Vis.P20.EnableIndex OF
		0..7:
			Vis.P20.Status[Vis.P20.EnableIndex]	:=	SHOW	;
	END_CASE

END_PROGRAM
```

### Program Logical/VisControl/HMIControl/ESRecover (IEC) - EStop Recovery Program

#### ESRecover.st - Cyclic code
```iecst
(********************************************************************
 * COPYRIGHT --
 ********************************************************************
 * Program: ESRecover
 * File: ESRecover.st
 * Author: NE
 ********************************************************************)

PROGRAM _CYCLIC

    //SET ESCLEAR BIT IF GLASS PRESENT AT ESTOP
	Control.ESClear := EMO.Recovery ;

	//DELAY SEAMING CONVEYORS RESTART AFTER ESTOP UNTIL GRINDING BELTS ALLOWED TO POSITION
	IF EDGENEG(Control.ESClear) THEN
		EMO.Latch1 := TRUE ;
		EMO.Latch2 := TRUE ;
	END_IF

	PresetSys.ESRestart[1] := LIMIT(10, PresetSys.ESRestart[1], 700) ;
	EMO.LatchTON1.IN := (EMO.Latch1) AND (SeamersII.DoneOUT[1]) ;
	EMO.LatchTON1.PT := PresetSys.ESRestart[1] ;
	EMO.LatchTON1 ();
	IF(EMO.LatchTON1.Q) THEN
		EMO.Latch1 := FALSE ;
	END_IF

	PresetSys.ESRestart[2] := LIMIT(10, PresetSys.ESRestart[2], 700) ;
	EMO.LatchTON2.IN := (EMO.Latch2) AND (SeamersII.DoneOUT[2]) ;
	EMO.LatchTON2.PT := PresetSys.ESRestart[2] ;
	EMO.LatchTON2 ();
	IF(EMO.LatchTON2.Q) THEN
		EMO.Latch2 := FALSE ;
	END_IF

	//AT ESTOP LATCH BIT TO ALLOW FOR MOVEMENT OF GLASS ON CONVEYORS AND PALLETS
	IF EDGEPOS(Control.EStop1) THEN
		EMO.StartLatch := TRUE ;
	END_IF

	EMO.Start.IN := EMO.StartLatch ;
	EMO.Start.PT := T#2s ;
	EMO.Start ();

	IF EDGEPOS(EMO.Start.Q) THEN
		EMO.StartLatch := FALSE ;
	END_IF

	//RESET ESCONFIRM BIT
	IF EDGEPOS(Control.EStop1) AND (Control.ESClear) OR EDGENEG(Control.ESClear) THEN
		EMO.Confirm[4] := FALSE ;
	END_IF

	//SWITCH TO EMO RECOVERY SCREEN IF ANY GLASS PRESENT
	IF EDGEPOS(Control.EStop1) AND NOT(Control.Empty) THEN
		Vis.P11.EnableIndex := 20 ;
		Vis.Page.New := P11_MIMIC ;
	END_IF

	//ESTOP RECOVERY SCREENS ACTIVE
	IF (Vis.P11.EnableIndex >= 20) AND (Vis.P11.EnableIndex <= 22) THEN
		EMO.Recovery := TRUE ;
	ELSE
		EMO.Recovery := FALSE ;
		Vis.EMO.Disp[0] := HIDE ;
		Vis.EMO.Disp[1] := HIDE ;
		Vis.EMO.Disp[2] := HIDE ;
		Vis.EMO.Disp[3] := HIDE ;
		Vis.EMO.Confirm[0] := FALSE ;
		Vis.EMO.Confirm[1] := FALSE ;
		Vis.EMO.Confirm[2] := FALSE ;
		Vis.EMO.Confirm[3] := FALSE ;
		Vis.EMO.Confirm[4] := FALSE ;
		Tracking00.Cleared := FALSE ;
		Tracking90.Cleared := FALSE ;
		Tracking01.Cleared := FALSE ;
		Tracking10.Cleared := FALSE ;
		Tracking91.Cleared := FALSE ;
		Tracking11.Cleared := FALSE ;
		Tracking20.Cleared := FALSE ;
		Tracking92.Cleared := FALSE ;
		Tracking30.Cleared := FALSE ;
		Tracking93.Cleared := FALSE ;
		Tracking40.Cleared := FALSE ;
		Tracking41.Cleared := FALSE ;
		Tracking50.Cleared := FALSE ;
		Tracking60.Cleared := FALSE ;
		Tracking70.Cleared := FALSE ;
		Tracking80.Cleared := FALSE ;
		Tracking81.Cleared := FALSE ;
		Tracking82.Cleared := FALSE ;
		Tracking51.Cleared := FALSE ;
	END_IF

	//RESET ALL BITS IF ESTOP PRESSED WHILE ON ESTOPSCREENS
	IF EDGEPOS(Control.EStop1) AND (EMO.Recovery) THEN
		Vis.EMO.Disp[0] := HIDE ;
		Vis.EMO.Disp[1] := HIDE ;
		Vis.EMO.Disp[2] := HIDE ;
		Vis.EMO.Disp[3] := HIDE ;
		Vis.EMO.Confirm[0] := FALSE ;
		Vis.EMO.Confirm[1] := FALSE ;
		Vis.EMO.Confirm[2] := FALSE ;
		Vis.EMO.Confirm[3] := FALSE ;
		Vis.EMO.Confirm[4] := FALSE ;
		Tracking00.Cleared := FALSE ;
		Tracking90.Cleared := FALSE ;
		Tracking01.Cleared := FALSE ;
		Tracking10.Cleared := FALSE ;
		Tracking91.Cleared := FALSE ;
		Tracking11.Cleared := FALSE ;
		Tracking20.Cleared := FALSE ;
		Tracking92.Cleared := FALSE ;
		Tracking30.Cleared := FALSE ;
		Tracking93.Cleared := FALSE ;
		Tracking40.Cleared := FALSE ;
		Tracking41.Cleared := FALSE ;
		Tracking50.Cleared := FALSE ;
		Tracking60.Cleared := FALSE ;
		Tracking70.Cleared := FALSE ;
		Tracking80.Cleared := FALSE ;
		Tracking81.Cleared := FALSE ;
		Tracking82.Cleared := FALSE ;
		Tracking51.Cleared := FALSE ;
	END_IF

	//ESTOP RECOVERY SCREEN CONFIRMATION AND CONTROLS
	CASE Vis.P11.EnableIndex OF
		//ESTOP SCREENS
		20:
			IF (Vis.EMO.Confirm[0]) THEN
				Vis.EMO.Disp[0] := SHOW ;
			END_IF
			IF (Vis.EMO.Confirm[1]) THEN
				Vis.EMO.Disp[1] := SHOW ;
			END_IF
			IF (Vis.EMO.Confirm[1]) AND (Control.Achieved1) THEN
				Vis.EMO.Disp[2] := SHOW;
			END_IF
		21:
			Vis.EMO.Disp[4] := SHOW ;
			IF (Vis.EMO.Confirm[2]) THEN
				Vis.EMO.Disp[3] := SHOW ;
				Vis.P11.EnableIndex := 22 ;
				Vis.EMO.Disp[4] := HIDE ;
				Vis.EMO.Confirm[4] := TRUE ;
			END_IF

			IF (Vis.EMO.Confirm[3]) THEN
				Tracking00.Cleared := FALSE ;
				Tracking90.Cleared := FALSE ;
				Tracking01.Cleared := FALSE ;
				Tracking10.Cleared := FALSE ;
				Tracking91.Cleared := FALSE ;
				Tracking11.Cleared := FALSE ;
				Tracking20.Cleared := FALSE ;
				Tracking92.Cleared := FALSE ;
				Tracking30.Cleared := FALSE ;
				Tracking93.Cleared := FALSE ;
				Tracking40.Cleared := FALSE ;
				Tracking41.Cleared := FALSE ;
				Tracking50.Cleared := FALSE ;
				Tracking60.Cleared := FALSE ;
				Tracking70.Cleared := FALSE ;
				Tracking80.Cleared := FALSE ;
				Tracking81.Cleared := FALSE ;
				Tracking82.Cleared := FALSE ;
				Tracking51.Cleared := FALSE ;
				Vis.EMO.Confirm[3] := FALSE ;
			END_IF
			//USE BITS SET FROM SCREEN TO CLEAR TRACKING DATA OF REMOVED PIECES
			Tracking00.ResES := FALSE ;
			Tracking90.ResES := FALSE ;
			Tracking01.ResES := FALSE ;
			Tracking10.ResES := FALSE ;
			Tracking91.ResES := FALSE ;
			Tracking11.ResES := FALSE ;
			Tracking20.ResES := FALSE ;
			Tracking92.ResES := FALSE ;
			Tracking30.ResES := FALSE ;
			Tracking93.ResES := FALSE ;
			Tracking40.ResES := FALSE ;
			Tracking41.ResES := FALSE ;
			Tracking50.ResES := FALSE ;
			Tracking60.ResES := FALSE ;
			Tracking70.ResES := FALSE ;
			Tracking80.ResES := FALSE ;
			Tracking81.ResES := FALSE ;
			Tracking82.ResES := FALSE ;
			Tracking51.ResES := FALSE ;
			IF EDGEPOS(Vis.EMO.Confirm[4]) THEN
				IF(Tracking00.Cleared) THEN
					Tracking00.ResES := TRUE ;
				END_IF
				IF(Tracking90.Cleared) THEN
					Tracking90.ResES := TRUE ;
				END_IF
				IF(Tracking01.Cleared) THEN
					Tracking01.ResES := TRUE ;
				END_IF
				IF(Tracking10.Cleared) THEN
					Tracking10.ResES := TRUE ;
				END_IF
				IF(Tracking91.Cleared) THEN
					Tracking91.ResES := TRUE ;
				END_IF
				IF(Tracking11.Cleared) THEN
					Tracking11.ResES := TRUE ;
				END_IF
				IF(Tracking20.Cleared) THEN
					Tracking20.ResES := TRUE ;
				END_IF
				IF(Tracking92.Cleared) THEN
					Tracking92.ResES := TRUE ;
				END_IF
				IF(Tracking30.Cleared) THEN
					Tracking30.ResES := TRUE ;
				END_IF
				IF(Tracking93.Cleared) THEN
					Tracking93.ResES := TRUE ;
				END_IF
				IF(Tracking40.Cleared) THEN
					Tracking40.ResES := TRUE ;
				END_IF
				IF(Tracking41.Cleared) THEN
					Tracking41.ResES := TRUE ;
				END_IF
				IF(Tracking50.Cleared) THEN
					Tracking50.ResES := TRUE ;
				END_IF
				IF(Tracking60.Cleared) THEN
					Tracking60.ResES := TRUE ;
				END_IF
				IF(Tracking70.Cleared) THEN
					Tracking70.ResES := TRUE ;
				END_IF
				IF(Tracking80.Cleared) THEN
					Tracking80.ResES := TRUE ;
				END_IF
				IF(Tracking81.Cleared) THEN
					Tracking81.ResES := TRUE ;
				END_IF
				IF(Tracking82.Cleared) THEN
					Tracking82.ResES := TRUE ;
				END_IF
				IF(Tracking51.Cleared) THEN
					Tracking51.ResES := TRUE ;
				END_IF

			END_IF

		22:
			//USE BITS SET FROM SCREEN TO CLEAR TRACKING DATA OF REMOVED PIECES
			Tracking00.ResES := FALSE ;
			Tracking90.ResES := FALSE ;
			Tracking01.ResES := FALSE ;
			Tracking10.ResES := FALSE ;
			Tracking91.ResES := FALSE ;
			Tracking11.ResES := FALSE ;
			Tracking20.ResES := FALSE ;
			Tracking92.ResES := FALSE ;
			Tracking30.ResES := FALSE ;
			Tracking93.ResES := FALSE ;
			Tracking40.ResES := FALSE ;
			Tracking41.ResES := FALSE ;
			Tracking50.ResES := FALSE ;
			Tracking60.ResES := FALSE ;
			Tracking70.ResES := FALSE ;
			Tracking80.ResES := FALSE ;
			Tracking81.ResES := FALSE ;
			Tracking82.ResES := FALSE ;
			Tracking51.ResES := FALSE ;
			Tracking00.Cleared := FALSE ;
			Tracking90.Cleared := FALSE ;
			Tracking01.Cleared := FALSE ;
			Tracking10.Cleared := FALSE ;
			Tracking91.Cleared := FALSE ;
			Tracking11.Cleared := FALSE ;
			Tracking20.Cleared := FALSE ;
			Tracking92.Cleared := FALSE ;
			Tracking30.Cleared := FALSE ;
			Tracking93.Cleared := FALSE ;
			Tracking40.Cleared := FALSE ;
			Tracking41.Cleared := FALSE ;
			Tracking50.Cleared := FALSE ;
			Tracking60.Cleared := FALSE ;
			Tracking70.Cleared := FALSE ;
			Tracking80.Cleared := FALSE ;
			Tracking81.Cleared := FALSE ;
			Tracking82.Cleared := FALSE ;
			Tracking51.Cleared := FALSE ;

	END_CASE

END_PROGRAM
```

### Program Logical/VisControl/HMIControl/Simulation (IEC) - Simulation control

#### Simulation.st - Cyclic code
```iecst
(********************************************************************
 * COPYRIGHT --
 ********************************************************************
 * Program: Simulation
 * File: Simulation.st
 * Author: NickE
 * Created: January 24, 2013
 ********************************************************************
 * Implementation of program Simulation
 ********************************************************************)

PROGRAM _INIT

	Control.EStop1 := TRUE ;
	Control.EStop2 := TRUE ;
	Simulation.Disp := SHOW ;
	Simulation.On := TRUE ;
	S100Reed.In := TRUE ;
	S102Reed.In := TRUE ;
	S104Reed.In := TRUE ;
	S106Reed.In := TRUE ;
	S108Reed.In := TRUE ;
	S110Reed.In := TRUE ;
	S112Reed.In := TRUE ;
	S114Reed.In := TRUE ;
	S120Reed.In := TRUE ;
	S122Reed.In := TRUE ;
	S124Reed.In := TRUE ;
	S126Reed.In := TRUE ;
	WashRun.In := TRUE ;
	CLB.Input.ETAD_02	:=	TRUE	;
	CRB.Input.ETAD_02	:=	TRUE	;

END_PROGRAM

PROGRAM _CYCLIC

	Ax1.OriginSet	:=	Control.Achieved1	;
	Ax1.Error		:=	FALSE				;
	Servo1POT.In	:= 	TRUE				;
	Servo1NOT.In	:=	TRUE				;
	Ax2.OriginSet	:=	Control.Achieved1	;
	Ax2.Error		:=	FALSE				;
	Servo2POT.In	:=	TRUE				;
	Servo2NOT.In	:=	TRUE				;

	IF EDGEPOS(Control.EStop2) THEN
		Control.EStop1	:=	TRUE	;
	END_IF

	IF NOT(TestAuto.In) THEN
		S30Reed.In	:= 	NOT(Sol30Pal1.Auto)	;
		S31Reed.In	:=	(Sol30Pal1.Auto)	;
		S32Reed.In	:= 	NOT(Sol31Pal2.Auto)	;
		S33Reed.In	:=	(Sol31Pal2.Auto)	;
		S34Reed.In	:= 	NOT(Sol32Pal3.Auto)	;
		S35Reed.In	:=	(Sol32Pal3.Auto)	;
		S36Reed.In	:= 	NOT(Sol33Pal4.Auto)	;
		S37Reed.In	:=	(Sol33Pal4.Auto)	;
		S52Reed.In	:= 	NOT(Sol40Datum.Auto);
		S53Reed.In	:=	(Sol40Datum.Auto)	;
	END_IF

END_PROGRAM
```

### Program Logical/VisControl/BatchDisp/BatchData (IEC) - Track Batching Data

#### BatchData.st - Implementation code
```iecst
(********************************************************************
 * COPYRIGHT --
 ********************************************************************
 * PROGRAM: BatchData
 * File: BatchData.st
 * Author: NickE
 ********************************************************************)

PROGRAM _INIT

	//HIDE OPTIONS SCREEN
	VisBatch.P1.Status[0]	:=	HIDE	;
	//SET DEFAULT COLOURS ON INITIAL POWER UP
	IF(CLPT2.Rev = 0) THEN
		CAPT.Clear	:=	GREY	;
		CAPT.Start	:=	RED	;
		CAPT.Slow	:=	14	;
		CLPT2.Rev	:=	1	;
	END_IF
	//SET IMPERIAL AS DEFAULT
	CAPT.Rev := 1 ;

END_PROGRAM

PROGRAM _CYCLIC

	DataFlow.IndexRow	:=	LIMIT(1,DataFlow.IndexRow,12);
	DataFlow.IndexLoad	:=	LIMIT(1,DataFlow.IndexLoad,12);

	//SCALE BATCH SIZE VALUES TO FULL HD SCREEN SIZE
	ScaleBatch.RefY1[0].x	:=	00.0	;
	ScaleBatch.RefY1[0].y	:=	00.0	;
	ScaleBatch.RefY1[1].x	:=	1000.0	;
	ScaleBatch.RefY1[1].y	:=	345.0	;	//SCALE VALUES TO PERCENTAGE OF ACTUAL SIZE
	ScaleBatch.ScaleY1.NoOfPoints	:=	2		;
	ScaleBatch.ScaleY1.ptr_table	:=	ADR(ScaleBatch.RefY1)	;

	ScaleBatch.RefWidth[0].x	:=	00.0	;
	ScaleBatch.RefWidth[0].y	:=	00.0	;
	ScaleBatch.RefWidth[1].x	:=	1000.0	;
	ScaleBatch.RefWidth[1].y	:=	345.0	;	//SCALE VALUES TO PERCENTAGE OF ACTUAL SIZE
	ScaleBatch.ScaleWidth.NoOfPoints	:=	2		;
	ScaleBatch.ScaleWidth.ptr_table	:=	ADR(ScaleBatch.RefWidth)	;

	ScaleBatch.RefLength[0].x	:=	00.0	;
	ScaleBatch.RefLength[0].y	:=	00.0	;
	ScaleBatch.RefLength[1].x	:=	1000.0	;
	ScaleBatch.RefLength[1].y	:=	345.0	;	//SCALE VALUES TO PERCENTAGE OF ACTUAL SIZE
	ScaleBatch.ScaleLength.NoOfPoints	:=	2		;
	ScaleBatch.ScaleLength.ptr_table	:=	ADR(ScaleBatch.RefLength)	;

	ScaleBatch.RefGapL[0].x	:=	00.0	;
	ScaleBatch.RefGapL[0].y	:=	00.0	;
	ScaleBatch.RefGapL[1].x	:=	1000.0	;
	ScaleBatch.RefGapL[1].y	:=	345.0	;	//SCALE VALUES TO PERCENTAGE OF ACTUAL SIZE
	ScaleBatch.ScaleGapL.NoOfPoints	:=	2		;
	ScaleBatch.ScaleGapL.ptr_table	:=	ADR(ScaleBatch.RefGapL)	;

	ScaleBatch.RefGapW[0].x	:=	00.0	;
	ScaleBatch.RefGapW[0].y	:=	00.0	;
	ScaleBatch.RefGapW[1].x	:=	1000.0	;
	ScaleBatch.RefGapW[1].y	:=	345.0	;	//SCALE VALUES TO PERCENTAGE OF ACTUAL SIZE
	ScaleBatch.ScaleGapW.NoOfPoints	:=	2		;
	ScaleBatch.ScaleGapW.ptr_table	:=	ADR(ScaleBatch.RefGapW)	;

	CASE VisBatch.State OF
		RESET_WAIT:
			//USE CONDITION TO RESET VALUES WHEN REQUIRED
			VisBatch.Param.fill		:=	15	;
			VisBatch.Param.color	:=	15	;
			VisBatch.Param.back		:=	255	;
			VisBatch.Param.font1		:=	13	;
			VisBatch.Param.fore1		:=	45	;
			VisBatch.Control.RowsIndex	:=	1	;
			VisBatch.Control.RowIndex	:=	0	;
			VisBatch.Control.LongestScaled	:=	0	;
			VisBatch.Control.LongestOld	:=	VisBatch.Control.LongestScaled	;
			VisBatch.Control.X1Old	:=	0	;
			VisBatch.Control.Y1Old	:=	0	;
			ScaleBatch.ScaleGapL.x	:=	LoadPerm.Gap	;
			ScaleBatch.ScaleGapL();
			VisBatch.Control.GapLScaled	:=	REAL_TO_UINT(ScaleBatch.ScaleGapL.y)	;
			ScaleBatch.ScaleGapW.x	:=	RowPerm.Gap	;
			ScaleBatch.ScaleGapW();
			VisBatch.Control.GapWScaled	:=	REAL_TO_UINT(ScaleBatch.ScaleGapW.y)	;
			VisBatch.P1.Index	:=	0	;
			IF EDGEPOS(X2X18.P16)THEN
				VisBatch.State := CONFIRM_LOAD;
			END_IF

		CONFIRM_LOAD:
			VisBatch.P1.Index	:=	3	;
			IF(VisBatch.API.READY <> 1) THEN
				VisBatch.API.VC_HANDLE := VA_Setup(1 , 'BatchP')	;

				IF(VisBatch.API.VC_HANDLE <> 0) THEN
					VisBatch.API.READY := 1	;
				END_IF
			END_IF

			//CLEAR SCREEN USING REDRAW
			IF(VisBatch.API.READY = 1) THEN
				IF(VA_Saccess(1,VisBatch.API.VC_HANDLE)= 0) THEN
					VA_Redraw(1,VisBatch.API.VC_HANDLE)	;
					VA_Srelease(1,VisBatch.API.VC_HANDLE)	;
					VisBatch.P1.EnableIndex	:=	0	;
				END_IF
			END_IF

			IF(Loads.Furnace9.NotEmpty) THEN
				FOR i := 0 TO 199 DO
					VisBatch.Displayed.Data[i]	:=	VisBatch.Displayed.Data[200]	;
				END_FOR
				VisBatch.Displayed.Index	:=	0	;
				Loads.FurnaceExit	:=	Loads.Furnace9	;
				Loads.Furnace9		:=	Loads.Furnace8	;
				Loads.Furnace8		:=	Loads.Furnace7	;
				Loads.Furnace7		:=	Loads.Furnace6	;
				Loads.Furnace6		:=	Loads.Furnace5	;
				Loads.Furnace5		:=	Loads.Furnace4	;
				Loads.Furnace4		:=	Loads.Furnace3	;
				Loads.Furnace3		:=	Loads.Furnace2	;
				Loads.Furnace2		:=	Loads.Furnace1	;
				Loads.Furnace1	:=	Loads.Empty	;
				VisBatch.State	:=	EXTRACT_VALUES	;
			ELSE
				VisBatch.State	:=	RESET_WAIT	;
				VisBatch.P1.EnableIndex	:=	0	;
			END_IF

		CONFIRM_CLEAR:
			VisBatch.State	:=	REDRAW	;

		EXTRACT_VALUES:

			VisBatch.P1.Index	:=	1	;
			CASE VisBatch.Control.RowIndex OF
				0:	//EXTRACT ROW WIDTH FROM .Row[0].Width AND INCREMENT .RowIndex
					VisBatch.Control.RowWidthRaw	:=	Loads.FurnaceExit.Rows[VisBatch.Control.RowsIndex].Row[0].Width	;
					VisBatch.Control.RowIndex	:=	1	;
					VisBatch.State	:=	CALCULATE_X1	;
				1..14:
					VisBatch.Control.RowIndex	:=	VisBatch.Control.RowIndex + 1	;
					VisBatch.State	:=	CALCULATE_X1	;
				15:	//MAX ROW NUMBER REACHED, INCREMENT .RowsIndex, EXTRACT NEXT ROW WIDTH, SET LONGEST FROM PREVIOUS ROW
					VisBatch.Control.RowsIndex	:=	VisBatch.Control.RowsIndex + 1	;
					VisBatch.Control.RowIndex	:=	0	;
					VisBatch.Control.LongestOld	:=	VisBatch.Control.LongestScaled	;
			END_CASE

//		CALCULATE_X1: //LANDSCAPE
//			CASE (REAL_TO_UINT(VisBatch.Control.RowWidthRaw)) OF
//				0:
//					VisBatch.State	:=	REFRESH	;
//				ELSE
//					CASE VisBatch.Control.RowIndex OF
//						1:
//							CASE VisBatch.Control.RowsIndex OF
//								1:
//									VisBatch.Param.x1	:=	81	;//BATCH DISPLAY AREA LEFT + 2
//									VisBatch.Control.X1Old	:=	81	;//BATCH DISPLAY AREA LEFT + 1
//								2..15:
//									VisBatch.Param.x1	:=	VisBatch.Control.X1Old + VisBatch.Control.LongestOld + VisBatch.Control.GapLScaled	;
//									VisBatch.Control.X1Old	:=	VisBatch.Param.x1	;
//								16:
//							END_CASE
//					END_CASE
//
//					VisBatch.State	:=	CHECK_NEXT	;
//			END_CASE
//
		CALCULATE_X1: //PORTRAIT
			CASE (REAL_TO_UINT(VisBatch.Control.RowWidthRaw)) OF
				0:
					VisBatch.State	:=	REFRESH	;
				ELSE
					ScaleBatch.ScaleY1.x	:=	VisBatch.Control.RowWidthRaw	;
					ScaleBatch.ScaleY1();
					VisBatch.Control.RowWidthScaled	:=	REAL_TO_UINT(ScaleBatch.ScaleY1.y)	;
					VisBatch.Control.WidthRaw	:=	Loads.FurnaceExit.Rows[VisBatch.Control.RowsIndex].Row[VisBatch.Control.RowIndex].Width	;
					ScaleBatch.ScaleWidth.x	:=	VisBatch.Control.WidthRaw	;
					ScaleBatch.ScaleWidth();
					VisBatch.Param.width	:=	REAL_TO_UINT(ScaleBatch.ScaleWidth.y)	;

					CASE VisBatch.Control.RowIndex OF
						1:
							VisBatch.Param.x1 := REAL_TO_UINT(540 + (VisBatch.Control.RowWidthScaled/2) - VisBatch.Param.width);
							VisBatch.Control.X1Old := VisBatch.Param.x1;
						2..12:
							VisBatch.Param.x1 := REAL_TO_UINT(VisBatch.Control.X1Old - VisBatch.Param.width - VisBatch.Control.GapWScaled);
							VisBatch.Control.X1Old := VisBatch.Param.x1;
					END_CASE

					VisBatch.State	:=	CHECK_NEXT	;
			END_CASE

		CHECK_NEXT:
			VisBatch.Control.LengthRaw	:=	Loads.FurnaceExit.Rows[VisBatch.Control.RowsIndex].Row[VisBatch.Control.RowIndex].Length	;
//			VisBatch.Control.WidthRaw	:=	Loads.FurnaceExit.Rows[VisBatch.Control.RowsIndex].Row[VisBatch.Control.RowIndex].Width	;
			CASE (REAL_TO_UINT(VisBatch.Control.LengthRaw)) OF
				0:
					VisBatch.Control.RowsIndex	:=	VisBatch.Control.RowsIndex + 1	;
					VisBatch.Control.RowIndex	:=	0	;
					VisBatch.Control.LongestOld	:=	VisBatch.Control.LongestScaled	;
					VisBatch.Control.LongestScaled	:=	0	;
					VisBatch.State	:=	EXTRACT_VALUES	;
				ELSE
					VisBatch.State	:=	CALCULATE_Y1	;
			END_CASE

		CALCULATE_Y1:
//			ScaleBatch.ScaleWidth.x	:=	VisBatch.Control.WidthRaw	;
//			ScaleBatch.ScaleWidth();
//			VisBatch.Param.width	:=	REAL_TO_UINT(ScaleBatch.ScaleWidth.y)	;

			ScaleBatch.ScaleLength.x	:=	VisBatch.Control.LengthRaw	;
			ScaleBatch.ScaleLength();
			VisBatch.Param.height	:=	REAL_TO_UINT(ScaleBatch.ScaleLength.y)	;

//			CASE VisBatch.Control.RowIndex OF
//				1:
//					ScaleBatch.ScaleY1.x	:=	VisBatch.Control.RowWidthRaw	;
//					ScaleBatch.ScaleY1();
//					VisBatch.Control.RowWidthScaled	:=	REAL_TO_UINT(ScaleBatch.ScaleY1.y)	;
////					VisBatch.Param.y1	:= ((884 - VisBatch.Control.RowWidthScaled)/2) + 64	;//((DisplayWindow.Height - xxx)/2) + DisplayWindow.Top + 2
//					VisBatch.Param.y1	:= 64 + (884/2) + ((VisBatch.Control.RowWidthScaled)/2) - VisBatch.Param.height	;//CALCULATION TO MIRROR DISPLAY
//					VisBatch.Control.Y1Old	:=	VisBatch.Param.y1	;
//				2..13:
//					ScaleBatch.ScaleY1.x	:=	VisBatch.Control.WidthRaw	;
//					ScaleBatch.ScaleY1();
//					VisBatch.Control.WidthScaled	:=	REAL_TO_UINT(ScaleBatch.ScaleY1.y)	;
////					VisBatch.Param.y1	:= VisBatch.Param.height + VisBatch.Control.GapWScaled + VisBatch.Control.Y1Old	;
//					VisBatch.Param.y1	:= VisBatch.Control.Y1Old - VisBatch.Param.height - VisBatch.Control.GapWScaled	;
//					VisBatch.Control.Y1Old	:=	VisBatch.Param.y1	;
//
//			END_CASE
			CASE VisBatch.Control.RowIndex OF
				1:
					CASE VisBatch.Control.RowsIndex OF
						1:
							VisBatch.Control.LongestScaled := REAL_TO_INT((Loads.FurnaceExit.Rows[VisBatch.Control.RowsIndex].Row[0].Length) * 0.345);
							VisBatch.Param.y1 := REAL_TO_UINT(1775 - VisBatch.Control.LongestScaled);
							VisBatch.Control.Y1Old := VisBatch.Param.y1;
						2..15:
							VisBatch.Control.LongestScaled := REAL_TO_INT((Loads.FurnaceExit.Rows[VisBatch.Control.RowsIndex].Row[0].Length) * 0.345);
							VisBatch.Param.y1 := REAL_TO_UINT(VisBatch.Control.Y1Old - VisBatch.Control.LongestScaled - VisBatch.Control.GapLScaled);
							VisBatch.Control.Y1Old := VisBatch.Param.y1;
					END_CASE
			END_CASE

//			IF(VisBatch.Param.height > VisBatch.Control.LongestScaled) THEN
//				VisBatch.Control.LongestScaled	:=	VisBatch.Param.height	;
//			END_IF
			CASE CAPT.Rev OF //METRIC OR ENGLISH
				0:
					VisBatch.Param.str	:=	REAL_TO_STRING(VisBatch.Control.LengthRaw)	;
					VisBatch.Param.str	:=	CONCAT(VisBatch.Param.str,' X ')	;
					VisBatch.Control.StrTemp	:=	REAL_TO_STRING(VisBatch.Control.WidthRaw)	;
					VisBatch.Param.str	:=	CONCAT(VisBatch.Param.str,VisBatch.Control.StrTemp)	;
				1:

					DispStrDecode.SixteenthStr := '' ;
					DispStrDecode.WholeInch := REAL_TO_INT(floor(VisBatch.Control.LengthRaw / 25.4)) ;
					DispStrDecode.WholeInchREAL := INT_TO_REAL(DispStrDecode.WholeInch) ;
					DispStrDecode.Remainder := (VisBatch.Control.LengthRaw - (DispStrDecode.WholeInchREAL * 25.4)) ;
					DispStrDecode.Sixteenth := (DispStrDecode.Remainder/ 1.5875) ;//(25.4*(1/16))) ;
					CASE REAL_TO_INT(DispStrDecode.Sixteenth * 10) OF
						0..4: //0/16
							DispStrDecode.SixteenthStr := '' ;
						5..14: //1/16
							DispStrDecode.SixteenthStr := ' 1/16' ;
						15..24: //2/16
							DispStrDecode.SixteenthStr := ' 1/8' ;
						25..34: //3/16
							DispStrDecode.SixteenthStr := ' 3/16' ;
						35..44: //4/16
							DispStrDecode.SixteenthStr := ' 1/4' ;
						45..54: //5/16
							DispStrDecode.SixteenthStr := ' 5/16' ;
						55..64: //6/16
							DispStrDecode.SixteenthStr := ' 3/8' ;
						65..74: //7/16
							DispStrDecode.SixteenthStr := ' 7/16' ;
						75..84: //8/16
							DispStrDecode.SixteenthStr := ' 1/2' ;
						85..94: //9/16
							DispStrDecode.SixteenthStr := ' 9/16' ;
						95..104: //10/16
							DispStrDecode.SixteenthStr := ' 5/8' ;
						105..114: //11/16
							DispStrDecode.SixteenthStr := ' 11/16' ;
						115..124: //12/16
							DispStrDecode.SixteenthStr := ' 3/4' ;
						125..134: //13/16
							DispStrDecode.SixteenthStr := ' 13/16' ;
						135..144: //14/16
							DispStrDecode.SixteenthStr := ' 7/8' ;
						145..154: //15/16
							DispStrDecode.SixteenthStr := ' 15/16' ;
						155..159: //16/16
							DispStrDecode.SixteenthStr := '' ;
							DispStrDecode.WholeInchREAL := DispStrDecode.WholeInchREAL + 1 ;
					END_CASE
					DispStrDecode.float_len := ftoa(DispStrDecode.WholeInchREAL, ADR(VisBatch.Param.str)) ;
					VisBatch.Param.str := CONCAT(VisBatch.Param.str, DispStrDecode.SixteenthStr) ;
					VisBatch.Param.str := CONCAT(VisBatch.Param.str, ' X ');
					DispStrDecode.SixteenthStr := '' ;
					DispStrDecode.WholeInch := REAL_TO_INT(floor(VisBatch.Control.WidthRaw / 25.4)) ;
					DispStrDecode.WholeInchREAL := INT_TO_REAL(DispStrDecode.WholeInch) ;
					DispStrDecode.Remainder := (VisBatch.Control.WidthRaw - (DispStrDecode.WholeInchREAL * 25.4)) ;
					DispStrDecode.Sixteenth := (DispStrDecode.Remainder/ 1.5875) ;//(25.4*(1/16))) ;
					CASE REAL_TO_INT(DispStrDecode.Sixteenth * 10) OF
						0..4: //0/16
							DispStrDecode.SixteenthStr := '' ;
						5..14: //1/16
							DispStrDecode.SixteenthStr := ' 1/16' ;
						15..24: //2/16
							DispStrDecode.SixteenthStr := ' 1/8' ;
						25..34: //3/16
							DispStrDecode.SixteenthStr := ' 3/16' ;
						35..44: //4/16
							DispStrDecode.SixteenthStr := ' 1/4' ;
						45..54: //5/16
							DispStrDecode.SixteenthStr := ' 5/16' ;
						55..64: //6/16
							DispStrDecode.SixteenthStr := ' 3/8' ;
						65..74: //7/16
							DispStrDecode.SixteenthStr := ' 7/16' ;
						75..84: //8/16
							DispStrDecode.SixteenthStr := ' 1/2' ;
						85..94: //9/16
							DispStrDecode.SixteenthStr := ' 9/16' ;
						95..104: //10/16
							DispStrDecode.SixteenthStr := ' 5/8' ;
						105..114: //11/16
							DispStrDecode.SixteenthStr := ' 11/16' ;
						115..124: //12/16
							DispStrDecode.SixteenthStr := ' 3/4' ;
						125..134: //13/16
							DispStrDecode.SixteenthStr := ' 13/16' ;
						135..144: //14/16
							DispStrDecode.SixteenthStr := ' 7/8' ;
						145..154: //15/16
							DispStrDecode.SixteenthStr := ' 15/16' ;
						155..159: //16/16
							DispStrDecode.SixteenthStr := '' ;
							DispStrDecode.WholeInchREAL := DispStrDecode.WholeInchREAL + 1 ;
					END_CASE
					DispStrDecode.float_len := ftoa(DispStrDecode.WholeInchREAL, ADR(VisBatch.Control.StrTemp)) ;
					VisBatch.Param.str := CONCAT(VisBatch.Param.str, VisBatch.Control.StrTemp) ;
					VisBatch.Param.str := CONCAT(VisBatch.Param.str, DispStrDecode.SixteenthStr) ;
//					VisBatch.Control.StrReal	:=	VisBatch.Control.LengthRaw * 100	;
//					VisBatch.Control.StrReal	:=	VisBatch.Control.StrReal / 25.4 ;
//					VisBatch.Control.StrInt		:=	TRUNC(VisBatch.Control.StrReal)	;
//					VisBatch.Control.StrReal	:=	INT_TO_REAL(VisBatch.Control.StrInt)	;
//					VisBatch.Param.str	:=	REAL_TO_STRING(VisBatch.Control.StrReal/100)	;
//					VisBatch.Param.str	:=	CONCAT(VisBatch.Param.str,' X ')	;
//					VisBatch.Control.StrReal	:=	VisBatch.Control.WidthRaw * 100	;
//					VisBatch.Control.StrReal	:=	VisBatch.Control.StrReal / 25.4 ;
//					VisBatch.Control.StrInt		:=	TRUNC(VisBatch.Control.StrReal)	;
//					VisBatch.Control.StrReal	:=	INT_TO_REAL(VisBatch.Control.StrInt)	;
//					VisBatch.Control.StrTemp	:=	REAL_TO_STRING(VisBatch.Control.StrReal/100)	;
//					VisBatch.Param.str	:=	CONCAT(VisBatch.Param.str,VisBatch.Control.StrTemp)	;
			END_CASE

			VisBatch.Displayed.Data[VisBatch.Displayed.Index].x1	:=	VisBatch.Param.x1	;
			VisBatch.Displayed.Data[VisBatch.Displayed.Index].y1	:=	VisBatch.Param.y1	;
			VisBatch.Displayed.Data[VisBatch.Displayed.Index].width	:=	VisBatch.Param.width	;
			VisBatch.Displayed.Data[VisBatch.Displayed.Index].height	:=	VisBatch.Param.height	;
			VisBatch.Displayed.Data[VisBatch.Displayed.Index].str	:=	VisBatch.Param.str	;
			VisBatch.Displayed.Index	:=	VisBatch.Displayed.Index + 1	;

			VisBatch.State	:=	EXTRACT_VALUES	;

		REDRAW:
			VisBatch.P1.Index	:=	3	;
			IF(VisBatch.API.READY <> 1) THEN
				VisBatch.API.VC_HANDLE := VA_Setup(1 , 'BatchP')	;

				IF(VisBatch.API.VC_HANDLE <> 0) THEN
					VisBatch.API.READY := 1	;
				END_IF
			END_IF

			//CLEAR SCREEN USING REDRAW
			IF(VisBatch.API.READY = 1) THEN
				IF(VA_Saccess(1,VisBatch.API.VC_HANDLE)= 0) THEN
					VA_Redraw(1,VisBatch.API.VC_HANDLE)	;
					VA_Srelease(1,VisBatch.API.VC_HANDLE)	;
					VisBatch.State	:=	RESET_WAIT	;
					VisBatch.P1.EnableIndex	:=	0	;
				END_IF
			END_IF

		REFRESH:
			VisBatch.P1.Index	:=	2	;
			IF(VisBatch.Displayed.RefreshIndex <= VisBatch.Displayed.Index) THEN
				VisBatch.Param.x1	:=	VisBatch.Displayed.Data[VisBatch.Displayed.RefreshIndex].x1;
				VisBatch.Param.y1	:=	VisBatch.Displayed.Data[VisBatch.Displayed.RefreshIndex].y1;
				VisBatch.Param.width	:=	VisBatch.Displayed.Data[VisBatch.Displayed.RefreshIndex].width;
				VisBatch.Param.height	:=	VisBatch.Displayed.Data[VisBatch.Displayed.RefreshIndex].height;
				//ADDED TO SWITCH DISPLAY DIRECTION 150216
				CASE CLPT2.Start OF
					1:
						VisBatch.Param.x1 := (1919 - VisBatch.Displayed.Data[VisBatch.Displayed.RefreshIndex].x1 - VisBatch.Param.width) ;//1919 = FIXED VALUE
						VisBatch.Param.y1	:=	(947 - (VisBatch.Displayed.Data[VisBatch.Displayed.RefreshIndex].y1 - 65) - VisBatch.Param.height) ;//943 = DISPLAY BOX TOP + HEIGHT - 2, 65 = TOP + 2
				END_CASE
				VisBatch.Param.str	:=	VisBatch.Displayed.Data[VisBatch.Displayed.RefreshIndex].str;
				VisBatch.State	:=	REFRESH_RECTANGLE	;
				VisBatch.Displayed.RefreshIndex	:=	VisBatch.Displayed.RefreshIndex + 1	;
			ELSE
				VisBatch.State	:=	RESET_WAIT	;
				VisBatch.Displayed.RefreshIndex	:=	0	;
				VisBatch.P1.EnableIndex	:=	0	;
			END_IF

		REFRESH_RECTANGLE:
			IF(VisBatch.API.READY <> 1) THEN
				VisBatch.API.VC_HANDLE := VA_Setup(1 , 'BatchP')	;

				IF(VisBatch.API.VC_HANDLE <> 0) THEN
					VisBatch.API.READY := 1	;
				END_IF
			END_IF

			//DRAW RECTANGLE BASED ON x1, y1(TOP LEFT), x2(WIDTH) AND y2(HEIGHT) VALUES. fill AND color VALUES TO BE PERMANENT VALUES (USE SPARE PERMANENT VALUES)
			IF(VisBatch.API.READY = 1) THEN
				IF(VA_Saccess(1,VisBatch.API.VC_HANDLE)= 0) THEN
					VisBatch.API.Status :=VA_Rect (1,VisBatch.API.VC_HANDLE,VisBatch.Param.x1,VisBatch.Param.y1,VisBatch.Param.width,VisBatch.Param.height,VisBatch.Param.fill,VisBatch.Param.color) ;
					VA_Srelease(1,VisBatch.API.VC_HANDLE)	;
					VisBatch.State	:=	REFRESH_TEXTOUT1	;
				END_IF
			END_IF

		REFRESH_TEXTOUT1:
			IF(VisBatch.API.READY <> 1) THEN
				VisBatch.API.VC_HANDLE := VA_Setup(1 , 'BatchP')	;

				IF(VisBatch.API.VC_HANDLE <> 0) THEN
					VisBatch.API.READY := 1	;
				END_IF
			END_IF

			IF(VisBatch.API.READY = 1) THEN
				IF(VA_Saccess(1,VisBatch.API.VC_HANDLE)= 0) THEN
					VA_Textout (1,VisBatch.API.VC_HANDLE,VisBatch.Param.font1,VisBatch.Param.x1,VisBatch.Param.y1,VisBatch.Param.fore1,VisBatch.Param.back,VisBatch.Param.str) ;
					VA_Srelease(1,VisBatch.API.VC_HANDLE)	;
					VisBatch.State	:=	REFRESH	;
				END_IF
			END_IF

	END_CASE

	//VISUALISATION CONTROLS
	//OPTIONS TEXT DISPLAY
	VisBatch.P1.Status[1]	:=	HIDE	;
	VisBatch.P1.Status[2]	:=	HIDE	;
	VisBatch.P1.Status[3]	:=	HIDE	;
	VisBatch.P1.Status[4]	:=	HIDE	;
	VisBatch.P1.Status[5]	:=	HIDE	;
	VisBatch.P1.Status[6]	:=	HIDE	;
	VisBatch.P1.Status[7]	:=	HIDE	;
	VisBatch.P1.Status[8]	:=	HIDE	;
	VisBatch.P1.Status[9]	:=	HIDE	;
	VisBatch.P1.Status[10]	:=	HIDE	;
	VisBatch.P1.Status[11]	:=	HIDE	;
	VisBatch.P1.Status[12]	:=	HIDE	;
	VisBatch.P1.Status[14]	:=	HIDE	;
	VisBatch.P1.Status[15]	:=	HIDE	;
	VisBatch.P1.Status[16]	:=	HIDE	;
	VisBatch.P1.Status[17]	:=	HIDE	;//ADDED TO SWITCH DISPLAY DIRECTION 150216
	VisBatch.P1.Status[18]	:=	HIDE	;//ADDED TO SWITCH DISPLAY DIRECTION 150216
	CASE CAPT.Slow OF
		11:
			CASE CLPT2.Clear OF
				0:
					VisBatch.P1.Status[1]	:= SHOW	;
				1:
					VisBatch.P1.Status[7]	:= SHOW	;
			END_CASE
		12:
			CASE CLPT2.Clear OF
				0:
					VisBatch.P1.Status[2]	:= SHOW	;
				1:
					VisBatch.P1.Status[8]	:= SHOW	;
			END_CASE
		13:
			CASE CLPT2.Clear OF
				0:
					VisBatch.P1.Status[3]	:= SHOW	;
				1:
					VisBatch.P1.Status[9]	:= SHOW	;
			END_CASE
		14:
			CASE CLPT2.Clear OF
				0:
					VisBatch.P1.Status[4]	:= SHOW	;
				1:
					VisBatch.P1.Status[10]	:= SHOW	;
			END_CASE
		15:
			CASE CLPT2.Clear OF
				0:
					VisBatch.P1.Status[5]	:= SHOW	;
				1:
					VisBatch.P1.Status[11]	:= SHOW	;
			END_CASE
		16:
			CASE CLPT2.Clear OF
				0:
					VisBatch.P1.Status[6]	:= SHOW	;
				1:
					VisBatch.P1.Status[12]	:= SHOW	;
			END_CASE
	END_CASE
	CASE CAPT.Start OF
		0:
			VisBatch.P1.Colour[0]	:=	BLACK	;
		1:
			VisBatch.P1.Colour[0]	:=	FONT_BLUE	;
		2:
			VisBatch.P1.Colour[0]	:=	FONT_GREEN	;
		4:
			VisBatch.P1.Colour[0]	:=	FONT_DARK_RED	;
		5:
			VisBatch.P1.Colour[0]	:=	FONT_MAGENTA	;
		7:
			VisBatch.P1.Colour[0]	:=	FONT_LIGHT_GREY	;
		8:
			VisBatch.P1.Colour[0]	:=	FONT_DARK_GREY	;
		11:
			VisBatch.P1.Colour[0]	:=	FONT_LIGHT_BLUE	;
		15:
			VisBatch.P1.Colour[0]	:=	FONT_WHITE	;
		42:
			VisBatch.P1.Colour[0]	:=	FONT_ORANGE	;
		45:
			VisBatch.P1.Colour[0]	:=	FONT_RED	;
		46:
			VisBatch.P1.Colour[0]	:=	FONT_YELLOW	;
	END_CASE
	CASE CLPT2.Clear OF
		0:	//GRAPHIC DISPLAY
			VisBatch.P1.Status[13]	:= SHOW	;
		1:	//LIST DISPLAY
			VisBatch.P1.Status[13]	:= HIDE	;
	END_CASE

	CASE VisBatch.P1.EnableIndex OF
		1:
			VisBatch.P1.Status[14]	:=	SHOW	;
		2:
			VisBatch.P1.Status[15]	:=	SHOW	;
	END_CASE

	CASE VisBatch.P1.Index OF
		1..5:
			VisBatch.P1.Status[16]	:=	SHOW	;
	END_CASE

	//ADDED TO SWITCH DISPLAY DIRECTION 150216
	CASE CLPT2.Start OF
		0:
			VisBatch.P1.Status[17]	:=	SHOW	;
		1:
			VisBatch.P1.Status[18]	:=	SHOW	;
	END_CASE

	IF(Loads.Furnace9.NotEmpty) THEN
		VisBatch.P1.Colour[1]	:=	BLUE	;
	ELSE
		VisBatch.P1.Colour[1]	:=	GREY	;
	END_IF
	IF(Loads.Furnace8.NotEmpty) THEN
		VisBatch.P1.Colour[2]	:=	BLUE	;
	ELSE
		VisBatch.P1.Colour[2]	:=	GREY	;
	END_IF
	IF(Loads.Furnace7.NotEmpty) THEN
		VisBatch.P1.Colour[3]	:=	BLUE	;
	ELSE
		VisBatch.P1.Colour[3]	:=	GREY	;
	END_IF
	IF(Loads.Furnace6.NotEmpty) THEN
		VisBatch.P1.Colour[4]	:=	BLUE	;
	ELSE
		VisBatch.P1.Colour[4]	:=	GREY	;
	END_IF
	IF(Loads.Furnace5.NotEmpty) THEN
		VisBatch.P1.Colour[5]	:=	BLUE	;
	ELSE
		VisBatch.P1.Colour[5]	:=	GREY	;
	END_IF
	IF(Loads.Furnace4.NotEmpty) THEN
		VisBatch.P1.Colour[6]	:=	BLUE	;
	ELSE
		VisBatch.P1.Colour[6]	:=	GREY	;
	END_IF
	IF(Loads.Furnace3.NotEmpty) THEN
		VisBatch.P1.Colour[7]	:=	BLUE	;
	ELSE
		VisBatch.P1.Colour[7]	:=	GREY	;
	END_IF
	IF(Loads.Furnace2.NotEmpty) THEN
		VisBatch.P1.Colour[8]	:=	BLUE	;
	ELSE
		VisBatch.P1.Colour[8]	:=	GREY	;
	END_IF
	IF(Loads.Furnace1.NotEmpty) THEN
		VisBatch.P1.Colour[9]	:=	BLUE	;
	ELSE
		VisBatch.P1.Colour[9]	:=	GREY	;
	END_IF

END_PROGRAM
```

### Program Logical/VisControl/ServiceControl/S_Level (IEC) - Password Level control

#### S_Level.st - Cyclic code
```iecst
(********************************************************************
 * COPYRIGHT --
 ********************************************************************
 * PROGRAM: S_Level
 * File: S_ServiceLevel.st
 * Author: nicke
 * Created: May 01, 2013
 ********************************************************************
 * Implementation OF PROGRAM S_Level
 ********************************************************************)

PROGRAM _INIT

	ServiceVis.API.VC_HANDLE	:=	0	;

END_PROGRAM

PROGRAM _CYCLIC

	CASE ServiceVis.Page.Current OF
		P00_INITIALIZE:
			//Init time - 3 sec
			ServiceVis.Init.TimeoutEnable	:= TRUE					;
			ServiceVis.Init.TON.IN			:= ServiceVis.Init.TimeoutEnable	;
			ServiceVis.Init.TON.PT			:= T#3000ms				;
			ServiceVis.Init.TON ();

			ServiceVis.Init.Progress	:=	UDINT_TO_USINT(TIME_TO_UDINT(ServiceVis.Init.TON.ET) / 30);
			IF (ServiceVis.Init.TON.Q) THEN
				//Switch to Menu Screen
				ServiceVis.Page.New			:= 	P10_MENU	;
				ServiceVis.Init.TimeoutEnable	:= 	FALSE		;
			END_IF
	END_CASE

	(*Hidden message control*)
	ServiceVis.Message.Display	;
	ServiceVis.Message.Text	;

	//GET TOUCH ACTION FROM SCREEN
	IF(ServiceVis.API.READY <> 1) THEN
		ServiceVis.API.VC_HANDLE := VA_Setup(1 , 'Servic')	;

		IF(ServiceVis.API.VC_HANDLE <> 0) THEN
			ServiceVis.API.READY := 1	;
		END_IF
	END_IF

	IF(ServiceVis.API.READY = 1) THEN
		IF(VA_Saccess(1,ServiceVis.API.VC_HANDLE)= 0) THEN
			VA_GetTouchAction (1,ServiceVis.API.VC_HANDLE,0,(ADR(ServiceVis.API.TOUCH))) ;
			VA_Srelease(1,ServiceVis.API.VC_HANDLE)	;
		END_IF
	END_IF

	IF(ServiceVis.API.TOUCH.status = 1) THEN
		ServiceLevel.ScreenTouch	:=	TRUE	;
	END_IF

	//PAGE CHANGE
	IF(ServiceVis.Page.Current <> ServiceVis.Page.Old) THEN
		ServiceVis.Page.Changed	:=	TRUE	;
	ELSE
		ServiceVis.Page.Changed	:=	FALSE	;
	END_IF
	ServiceVis.Page.Old	:=	ServiceVis.Page.Current;

	//HIDE DROP DOWN SCREENS
	IF(ServiceVis.Page.Changed) THEN
		ServiceVis.Start.Enable	:=	HIDE	;
		ServiceVis.IP.Enable		:=	HIDE	;
		ServiceVis.Status.Enable	:=	HIDE	;
		ServiceLevel.Enable	:=	HIDE	;
		ServiceLevel.EnableSup	:=	HIDE	;
		ServiceLevel.EnableEng	:=	HIDE	;
		ServiceLevel.EnableTech	:=	HIDE	;
		IF NOT(Control.ESClear) THEN
			ServiceVis.P11.EnableIndex		:=	24	;
		END_IF
		ServiceVis.P12.EnableIndex		:=	24	;
	END_IF

	//HEADER BAR COLOUR DISPLAY
	CASE ServiceVis.Page.Current OF
		P10_MENU:
			ServiceVis.HeaderColour	:=	RED_MENU	;
		P11_MIMIC:
			ServiceVis.HeaderColour	:=	GREY_MIMIC	;
		P12_OPTIONS:
			ServiceVis.HeaderColour	:=	GREEN_OPTIONS	;
		P13_SETTINGS:
			ServiceVis.HeaderColour	:=	BLUE	;
		P14_DRIVES:
			ServiceVis.HeaderColour	:=	VIOLET	;
		P15_SERVOS:
			ServiceVis.HeaderColour	:=	GREEN1	;
		P16_RIO:
			ServiceVis.HeaderColour	:=	LIGHTBLUE	;
		P17_ALARM:
			ServiceVis.HeaderColour	:=	RED	;
		P18_WARNING:
			ServiceVis.HeaderColour	:=	ORANGE	;
		P19_EVENT:
			ServiceVis.HeaderColour	:=	YELLOW_EVENT	;
		P20_ASHTON_TECH:
			ServiceVis.HeaderColour	:=	GREY_ASHTON	;
		P21_SDM:
			ServiceVis.HeaderColour	:=	ORANGE_SDM	;
		P30_VARIABLES:
			Vis.HeaderColour	:=	LILAC	;
	END_CASE

	//RESET SYSTEM PASSWORD
	IF NOT(SysPerm.PasswordDefault) THEN
		SysPerm.Password[0]		:= 	''		;
		SysPerm.Password[1]		:= 	'1'		;
		SysPerm.Password[2]		:= 	'5'		;
		SysPerm.Password[3]		:= 	'4046'	;
		SysPerm.PasswordDefault	:= 	TRUE	;
		ServiceLevel.Delay.IN			:=	TRUE	;
		ServiceLevel.Enable			:=	HIDE	;
		ServiceLevel.ResetEnable		:=	SHOW	;
	END_IF

	//ENABLE SUPERVISOR LEVEL FOR TESTING
	ServiceLevel.Level	:=	LIMIT(3,ServiceLevel.Level,3)	;

	//	//Password control. Use level to enable different layers on screen rather than seperate screens.
	CASE ServiceLevel.Level OF
		//		OPERATOR:
		//			ServiceLevel.SupResetStart			:=	FALSE	;
		//			ServiceLevel.EngResetStart			:=	FALSE	;
		//			ServiceLevel.TechResetStart		:=	FALSE	;
		//			ServiceLevel.EnableSup				:=	HIDE	;
		//			ServiceLevel.EnableEng				:=	HIDE	;
		//			ServiceLevel.EnableTech			:=	HIDE	;
		//			ServiceLevel.GTOperatorEnable		:=	HIDE	;
		//			ServiceLevel.GTSupervisorEnable	:=	HIDE	;
		//			ServiceLevel.GTEngineerEnable		:=	HIDE	;
		//			ServiceLevel.TestMode				:=	HIDE	;
		//			Control.Test				:=	FALSE	;
		//			ServiceLevel.TestModeEnable		:=	HIDE	;
		//		SUPERVISOR:
		//			ServiceLevel.SupResetStart			:=	TRUE	;
		//			ServiceLevel.EnableSup				:=	ServiceLevel.Enable	;
		//			ServiceLevel.EnableEng				:=	HIDE	;
		//			ServiceLevel.EnableTech			:=	HIDE	;
		//			ServiceLevel.GTOperatorEnable		:=	SHOW	;
		//			ServiceLevel.GTSupervisorEnable	:=	HIDE	;
		//			ServiceLevel.GTEngineerEnable		:=	HIDE	;
		//			ServiceLevel.TestMode				:=	HIDE	;
		//			Control.Test				:=	FALSE	;
		//			ServiceLevel.TestModeEnable		:=	HIDE	;
		//		ENGINEER:
		//			ServiceLevel.EngResetStart			:=	TRUE	;
		//			ServiceLevel.EnableSup				:=	HIDE	;
		//			ServiceLevel.EnableEng				:=	ServiceLevel.Enable	;
		//			ServiceLevel.EnableTech			:=	HIDE	;
		//			ServiceLevel.GTOperatorEnable		:=	SHOW	;
		//			ServiceLevel.GTSupervisorEnable	:=	SHOW	;
		//			ServiceLevel.GTEngineerEnable		:=	HIDE	;
		//			ServiceLevel.TestMode				:=	HIDE	;
		//			ServiceLevel.TestModeEnable		:=	HIDE	;
		//			IF(Control.Empty) AND(Control.Achieved) THEN
		//				ServiceLevel.TestMode	:=	SHOW	;
		//			END_IF
		//			IF(Control.Test)THEN
		//				ServiceLevel.TestModeEnable	:=	SHOW	;
		//				ServiceLevel.TestMode	:=	SHOW	;
		//			END_IF
		ASHTON_TECH:
			ServiceLevel.TechResetStart		:=	TRUE	;
			ServiceLevel.EnableSup				:=	HIDE	;
			ServiceLevel.EnableEng				:=	HIDE	;
			ServiceLevel.EnableTech			:=	ServiceLevel.Enable	;
			ServiceLevel.GTOperatorEnable		:=	SHOW	;
			ServiceLevel.GTSupervisorEnable	:=	SHOW	;
			ServiceLevel.GTEngineerEnable		:=	SHOW	;
			ServiceLevel.TestMode				:=	HIDE	;
			ServiceLevel.TestModeEnable		:=	HIDE	;
			IF(Control.Empty) AND(Control.Achieved1) THEN
				ServiceLevel.TestMode	:=	SHOW	;
			END_IF
			IF(Control.Test)THEN
				ServiceLevel.TestModeEnable	:=	SHOW	;
				ServiceLevel.TestMode	:=	SHOW	;
			END_IF
	END_CASE

	//RESET DROP DOWN SCREENS WHEN PASSWORD DISPLAYED
	IF EDGEPOS(ServiceLevel.Enable = SHOW) THEN
		ServiceVis.Start.Enable	:=	HIDE	;
		ServiceVis.IP.Enable		:=	HIDE	;
		ServiceVis.Status.Enable	:=	HIDE	;
	END_IF

	//	//ScreenTouch control for cancel password delay.
	//	ServiceLevel.SupDelay.IN	:=	(ServiceLevel.SupResetStart) AND NOT(ServiceLevel.ScreenTouch)	;
	//	ServiceLevel.SupDelay.PT	:=	t#2m	;
	//	ServiceLevel.SupDelay();
	//
	//	IF EDGEPOS(ServiceLevel.SupDelay.Q) THEN
	//		ServiceLevel.Level	:=	0	;
	//	END_IF
	//
	//	ServiceLevel.EngDelay.IN	:=	(ServiceLevel.EngResetStart) AND NOT(ServiceLevel.ScreenTouch) AND NOT(ServiceLevel.BlockEng)	;
	//	ServiceLevel.EngDelay.PT	:=	t#2m	;
	//	ServiceLevel.EngDelay();
	//
	//	IF EDGEPOS(ServiceLevel.EngDelay.Q) THEN
	//		ServiceLevel.Level	:=	0	;
	//	END_IF
	//
	//	ServiceLevel.TechDelay.IN	:=	(ServiceLevel.TechResetStart) AND NOT(ServiceLevel.ScreenTouch) AND NOT(ServiceLevel.BlockTech)	;
	//	ServiceLevel.TechDelay.PT	:=	t#2m	;
	//	ServiceLevel.TechDelay();
	//
	//	IF EDGEPOS(ServiceLevel.TechDelay.Q) THEN
	//		ServiceLevel.Level	:=	0	;
	//	END_IF
	//
	ServiceLevel.ScreenTouch	:=	FALSE	;
	//
	//	IF(Control.Test) THEN
	//		ServiceLevel.BlockEng	:=	TRUE	;
	//		ServiceLevel.BlockTech	:=	TRUE	;
	//	ELSE
	//		ServiceLevel.BlockEng	:=	FALSE	;
	//		ServiceLevel.BlockTech	:=	FALSE	;
	//	END_IF
	//
	//	IF(ServiceVis.Page.Current = P20_ASHTON_TECH) OR(ServiceVis.Page.Current = P21_SDM) THEN
	//		ServiceLevel.BlockTech	:=	TRUE	;
	//	ELSE
	//		ServiceLevel.BlockTech	:=	FALSE	;
	//	END_IF
	//
	//	IF(Control.Achieved) AND(Control.Empty) THEN
	//		ServiceLevel.EngRefused	:=	HIDE	;
	//	END_IF
	//
	//	IF(ServiceLevel.RefusedConfirm) THEN
	//		ServiceLevel.EngRefused	:=	HIDE	;
	//		ServiceLevel.Enable		:=	HIDE	;
	//	END_IF
	//
	//	(*Change Password*)
	//	IF (ServiceLevel.SupConfirm) THEN
	//		SysPerm.Password[1]	:= 	ServiceLevel.SupNew	;
	//		ServiceLevel.Delay.IN	:=	TRUE			;
	//		ServiceLevel.SupEnable	:=	SHOW			;
	//	END_IF
	//
	//	IF (ServiceLevel.EngConfirm) THEN
	//		SysPerm.Password[2]	:= 	ServiceLevel.EngNew	;
	//		ServiceLevel.Delay.IN	:=	TRUE			;
	//		ServiceLevel.EngEnable	:=	SHOW			;
	//	END_IF
	//
	//	ServiceLevel.Delay.PT	:=	T#2000ms	;
	//	ServiceLevel.Delay ();
	//
	//	IF(ServiceLevel.Delay.Q) THEN
	//		ServiceLevel.SupConfirm	:= 	FALSE	;
	//		ServiceLevel.EngConfirm	:= 	FALSE	;
	//		ServiceLevel.SupNew		:= 	''		;
	//		ServiceLevel.EngNew		:= 	''		;
	//		ServiceLevel.SupEnable		:=	HIDE	;
	//		ServiceLevel.EngEnable		:=	HIDE	;
	//		ServiceLevel.ResetEnable	:=	HIDE	;
	//		ServiceLevel.Enable		:= 	HIDE	;
	//		ServiceLevel.Delay.IN		:=	FALSE	;
	//	END_IF
	//
	//	IF (ServiceLevel.Entered) THEN
	//		ServiceLevel.Enable	:= 	HIDE	;
	//		ServiceLevel.Entered	:= 	FALSE	;
	//	END_IF

END_PROGRAM
```

### Program Logical/VisControl/ServiceControl/S_Status (IEC) - Status Bar control

#### S_Status.st - Cyclic code
```iecst
(********************************************************************
 * COPYRIGHT --
 ********************************************************************
 * Program: S_Status
 * File: S_Status.st
 * Author: nicke
 * Created: May 02, 2013
 ********************************************************************
 * Implementation of program S_Status
 ********************************************************************)

PROGRAM _CYCLIC

	//SEAMER CONTROL SYSTEM STATUS
	IF NOT(Control.Achieved1) THEN
		ServiceVis.Status.StatusSeamer	:=	YELLOW		;
	END_IF

	IF(Control.Achieved1) THEN
		ServiceVis.Status.StatusSeamer	:=	GREEN	;
	END_IF

	IF(Pause.Active) THEN
		ServiceVis.Status.StatusSeamer	:=	ServiceVis.Status.GrnLmp	;
	END_IF

	IF(Control.ESClear) THEN
		ServiceVis.Status.StatusSeamer	:=	BLUE	;
	END_IF

	//NUMBER OF ACTIVE WARNINGS
	ServiceVis.Status.WarningCount		:=	0		;

	IF(Control.Warning) THEN
		ServiceVis.Status.StatusSeamer	:=	ORANGE	;
		ServiceVis.Status.WarningEnable	:=	SHOW	;
		FOR i:= 0 TO USINT_TO_INT(Warn.iMax) DO
			IF(Warn.Timeout[i]) THEN
				ServiceVis.Status.WarningCount	:=	ServiceVis.Status.WarningCount + 1	;
			END_IF
		END_FOR
	ELSE
		ServiceVis.Status.WarningEnable	:=	HIDE	;
		ServiceVis.Status.WarningCount		:=	0		;
	END_IF

	//NUMBER OF ACTIVE ALARMS
	ServiceVis.Status.AlarmCount	:=	0		;

	IF(Control.Alarm) THEN
		ServiceVis.Status.StatusSeamer	:=	RED		;
		ServiceVis.Status.AlarmEnable	:=	SHOW	;
		FOR i := 0 TO 60 DO
			IF(SysTemp.Alarms[i]) THEN
				ServiceVis.Status.AlarmCount	:=	ServiceVis.Status.AlarmCount + 1	;
			END_IF
		END_FOR
	ELSE
		ServiceVis.Status.AlarmEnable	:=	HIDE	;
		ServiceVis.Status.AlarmCount	:=	0		;
	END_IF

	//SERVO STATUS
	IF NOT(Ax1.Error) AND NOT(Ax2.Error) AND NOT(Ax3.Error) THEN
		ServiceVis.Status.StatusServo	:=	GREEN	;
	ELSE
		ServiceVis.Status.StatusServo	:=	YELLOW	;
	END_IF
	IF(Ax1.Error) OR(Ax2.Error) OR(Ax3.Error) THEN
		ServiceVis.Status.StatusServo	:=	RED	;
	END_IF

	//LASER STATUS
	IF(S56Lever.In) THEN
		ServiceVis.Status.StatusLaser	:=	GREEN	;
	ELSE
		ServiceVis.Status.StatusLaser	:=	YELLOW	;
	END_IF

	//LIGHTSTACK COLOURS
	IF(Control.RedLmp) THEN
		ServiceVis.Status.RedLmp	:=	RED		;
		ServiceVis.Status.TextRed	:=	1		;
	ELSE
		ServiceVis.Status.RedLmp	:=	GREY	;
		ServiceVis.Status.TextRed	:=	0		;
	END_IF

	IF(Control.GrnLmp) THEN
		ServiceVis.Status.GrnLmp	:=	GREEN	;
		ServiceVis.Status.TextGrn	:=	1		;
		IF(Pause.Active) THEN
			ServiceVis.Status.TextGrn	:=	2	;
		END_IF
	ELSE
		ServiceVis.Status.GrnLmp	:=	GREY	;
		ServiceVis.Status.TextGrn	:=	0		;
		IF(Pause.Active) THEN
			ServiceVis.Status.TextGrn	:=	2	;
		END_IF
	END_IF

	IF(Control.YelLmp) THEN
		ServiceVis.Status.YelLmp	:=	BLUE	;
		ServiceVis.Status.TextYel	:=	1		;
	ELSE
		ServiceVis.Status.YelLmp	:=	GREY	;
		ServiceVis.Status.TextYel	:=	0		;
	END_IF

	//RESET DROP DOWN SCREENS WHEN STATUS DISPLAYED
	IF EDGEPOS(ServiceVis.Status.Enable = SHOW) THEN
		ServiceVis.Start.Enable	:=	HIDE	;
		ServiceVis.IP.Enable		:=	HIDE	;
		ServiceLevel.Enable	:=	HIDE	;
		ServiceLevel.EnableSup	:=	HIDE	;
		ServiceLevel.EnableEng	:=	HIDE	;
		ServiceLevel.EnableTech	:=	HIDE	;
	END_IF

END_PROGRAM
```

### Program Logical/VisControl/ServiceControl/S_Start (IEC) - Start Visual controls

#### S_Start.st - Cyclic code
```iecst
(********************************************************************
 * COPYRIGHT --
 ********************************************************************
 * Program: S_Start
 * File: S_Start.st
 * Author: nicke
 * Created: May 02, 2013
 ********************************************************************
 * Implementation of program S_Start
 ********************************************************************)

PROGRAM _CYCLIC

	ServiceVis.Start.ResetEnable	:= HIDE	;

	//STATUS LIGHTS FOR SEAMER 1
	IF(Seamers.AutoStart[1]) THEN
		ServiceVis.Start.StatusSeam1	:=	GREEN	;
	ELSE
		ServiceVis.Start.StatusSeam1	:=	GREEN_DARK	;
	END_IF

	IF(Seamers.Enable[1]) AND NOT(Seamers.AutoStart[1]) THEN
		ServiceVis.Start.StatusSeam1	:=	YELLOW	;
	END_IF

	IF(MS1Belt1.Trip) THEN
		ServiceVis.Start.StatusSeam1	:=	RED	;
	ELSIF(MS2Belt2.Trip) THEN
		ServiceVis.Start.StatusSeam1	:=	RED	;
	ELSIF(MS3Belt3.Trip) THEN
		ServiceVis.Start.StatusSeam1	:=	RED	;
	ELSIF(MS4Belt4.Trip) THEN
		ServiceVis.Start.StatusSeam1	:=	RED	;
	ELSIF(MS9Vac1.Trip) THEN
		ServiceVis.Start.StatusSeam1	:=	RED	;
	ELSIF(MS11Vac3.Trip) THEN
		ServiceVis.Start.StatusSeam1	:=	RED	;
	ELSIF(MS23Vac5.Trip) THEN
		ServiceVis.Start.StatusSeam1	:=	RED	;
	ELSIF(MS24Vac6.Trip) THEN
		ServiceVis.Start.StatusSeam1	:=	RED	;
	END_IF

	//STATUS LIGHTS FOR SEAMER 2
	IF(Seamers.AutoStart[2]) THEN
		ServiceVis.Start.StatusSeam2	:=	GREEN	;
	ELSE
		ServiceVis.Start.StatusSeam2	:=	GREEN_DARK	;
	END_IF

	IF(Seamers.Enable[2]) AND NOT(Seamers.AutoStart[2]) THEN
		ServiceVis.Start.StatusSeam2	:=	YELLOW	;
	END_IF

	IF(MS5Belt5.Trip) THEN
		ServiceVis.Start.StatusSeam2	:=	RED	;
	ELSIF(MS6Belt6.Trip) THEN
		ServiceVis.Start.StatusSeam2	:=	RED	;
	ELSIF(MS7Belt7.Trip) THEN
		ServiceVis.Start.StatusSeam2	:=	RED	;
	ELSIF(MS8Belt8.Trip) THEN
		ServiceVis.Start.StatusSeam2	:=	RED	;
	ELSIF(MS10Vac2.Trip) THEN
		ServiceVis.Start.StatusSeam2	:=	RED	;
	ELSIF(MS12Vac4.Trip) THEN
		ServiceVis.Start.StatusSeam2	:=	RED	;
	ELSIF(MS25Vac7.Trip) THEN
		ServiceVis.Start.StatusSeam2	:=	RED	;
	ELSIF(MS26Vac8.Trip) THEN
		ServiceVis.Start.StatusSeam2	:=	RED	;
	END_IF

	IF EDGEPOS(Control.EStop1) AND(Control.Test) THEN
		ServiceVis.Start.Enable	:=	HIDE	;
	END_IF

END_PROGRAM
```

### Program Logical/VisControl/ServiceControl/S_Page10 (IEC) - Menu screen control

#### S_Page10.st - Cyclic code
```iecst
(********************************************************************
 * COPYRIGHT --
 ********************************************************************
 * Program: S_Page10
 * File: S_Page10.st
 * Author: nicke
 * Created: May 02, 2013
 ********************************************************************
 * Implementation of program S_Page10
 ********************************************************************)

PROGRAM _CYCLIC

	//MENU SCREEN
	ServiceVis.P10.Status[0]	:=	HIDE	;
	ServiceVis.P10.Status[1]	:=	HIDE	;
	ServiceVis.P10.Status[2]	:=	HIDE	;
	ServiceVis.P10.Status[3]	:=	HIDE	;
	ServiceVis.P10.Status[4]	:=	HIDE	;
	ServiceVis.P10.Status[5]	:=	HIDE	;
	ServiceVis.P10.Status[6]	:=	HIDE	;
	ServiceVis.P10.Status[7]	:=	HIDE	;
	ServiceVis.P10.Status[8]	:=	HIDE	;
	ServiceVis.P10.Status[9]	:=	HIDE	;
	ServiceVis.P10.Status[10]	:=	HIDE	;

	CASE ServiceVis.P10.EnableIndex OF
		0:
			ServiceVis.P10.Status[0]	:=	SHOW	;
		1:
			ServiceVis.P10.Status[1]	:=	SHOW	;
		2:
			ServiceVis.P10.Status[2]	:=	SHOW	;
		3:
			ServiceVis.P10.Status[3]	:=	SHOW	;
		4:
			ServiceVis.P10.Status[4]	:=	SHOW	;
		5:
			ServiceVis.P10.Status[5]	:=	SHOW	;
		6:
			ServiceVis.P10.Status[6]	:=	SHOW	;
		7:
			ServiceVis.P10.Status[7]	:=	SHOW	;
		8:
			ServiceVis.P10.Status[8]	:=	SHOW	;
		9:
			ServiceVis.P10.Status[9]	:=	SHOW	;

	END_CASE

END_PROGRAM
```

### Program Logical/VisControl/ServiceControl/S_Page11 (IEC) - Mimic screen control

#### S_Page11.st - Cyclic code
```iecst
(********************************************************************
 * COPYRIGHT --
 ********************************************************************
 * Program: S_Page11
 * File: S_Page11.st
 * Author: nicke
 * Created: May 02, 2013
 ********************************************************************
 * Implementation of program S_Page11
 ********************************************************************)

PROGRAM _CYCLIC

    //MIMIC SCREEN
    memcpy(ADR(ServiceVis.P11.Status),ADR(ServiceVis.HideAll),SIZEOF(ServiceVis.HideAll));
    memcpy(ADR(ServiceVis.P11.Status1),ADR(ServiceVis.HideAll),SIZEOF(ServiceVis.HideAll));
    //DISPLAY TRACK BLOCK CONDITION CONTROL
    ServiceVis.P11.Layers.Layer1 := HIDE ;
    ServiceVis.P11.Layers.Layer2 := HIDE ;
    ServiceVis.P11.Layers.Layer3 := HIDE ;
    ServiceVis.P11.Layers.Layer4 := HIDE ;
    ServiceVis.P11.Layers.Layer5 := HIDE ;
    ServiceVis.P11.Layers.Layer6 := HIDE ;
    ServiceVis.P11.Layers.Layer7 := HIDE ;
    ServiceVis.P11.Layers.Layer8 := HIDE ;
    ServiceVis.P11.Layers.Layer9 := HIDE ;
    ServiceVis.P11.Layers.Layer10 := HIDE ;
    ServiceVis.P11.Layers.Layer11 := HIDE ;
    ServiceVis.P11.Layers.Layer12 := HIDE ;
    ServiceVis.P11.Layers.Layer13 := HIDE ;
    ServiceVis.P11.Layers.Layer14 := HIDE ;
    ServiceVis.P11.Layers.Layer15 := HIDE ;

    CASE ServiceVis.P11.EnableIndex OF
		0:
			ServiceVis.P11.Status[0] := SHOW ;
			IF(ServiceLevel.Level > OPERATOR) AND(Tracking20.Busy) THEN
				ServiceVis.P11.Status1[0] := SHOW ;
			END_IF
			IF(Track208.Active) AND(Tracking20.Blocked) THEN
				ServiceVis.P11.Layers.Layer1 := SHOW ;
			END_IF
		1:
			ServiceVis.P11.Status[1] := SHOW ;
			IF(ServiceLevel.Level > OPERATOR) AND(Tracking30.Busy) THEN
				ServiceVis.P11.Status1[1] := SHOW ;
			END_IF
			IF(Track302.Active) AND(Tracking30.Blocked) THEN
				ServiceVis.P11.Layers.Layer2 := SHOW ;
			END_IF
		2:
			ServiceVis.P11.Status[2] := SHOW ;
			IF(ServiceLevel.Level > OPERATOR) AND(Tracking40.Busy) THEN
				ServiceVis.P11.Status1[2] := SHOW ;
			END_IF
			IF(Track402.Active) AND(Tracking40.Blocked) THEN
				ServiceVis.P11.Layers.Layer3 := SHOW ;
			END_IF
			IF(ServiceLevel.Level > OPERATOR) AND(Tracking41.Busy) THEN
				ServiceVis.P11.Status1[3] := SHOW ;
			END_IF
		3:
			ServiceVis.P11.Status[3] := SHOW ;
			IF(ServiceLevel.Level > OPERATOR) AND(Tracking50.Busy) THEN
				ServiceVis.P11.Status1[4] := SHOW ;
			END_IF
			IF(ServiceLevel.Level > OPERATOR) AND(Tracking80.Busy) THEN
				ServiceVis.P11.Status1[5] := SHOW ;
			END_IF
		4:
			ServiceVis.P11.Status[4] := SHOW ;
			IF(ServiceLevel.Level > OPERATOR) AND(Tracking60.Busy) THEN
				ServiceVis.P11.Status1[6] := SHOW ;
			END_IF
			IF(Track603.Active) AND(Tracking60.Blocked) THEN
				ServiceVis.P11.Layers.Layer4 := SHOW ;
			END_IF
			IF(ServiceLevel.Level > OPERATOR) AND(Tracking70.Busy) THEN
				ServiceVis.P11.Status1[7] := SHOW ;
			END_IF
			IF(ServiceLevel.Level > OPERATOR) AND(Tracking81.Busy) THEN
				ServiceVis.P11.Status1[8] := SHOW ;
			END_IF
			IF(Track812.Active) AND(Tracking81.Blocked) THEN
				ServiceVis.P11.Layers.Layer5 := SHOW ;
			END_IF
			IF(ServiceLevel.Level > OPERATOR) AND(Tracking82.Busy) THEN
				ServiceVis.P11.Status1[9] := SHOW ;
			END_IF
		5:
			ServiceVis.P11.Status[5] := SHOW ;
			IF(ServiceLevel.Level > OPERATOR) AND(Tracking00.Busy) THEN
				ServiceVis.P11.Status1[10] := SHOW ;
			END_IF
			IF(Track005.Active) AND(Tracking00.Blocked) THEN
				ServiceVis.P11.Layers.Layer6 := SHOW ;
			END_IF
			IF(Track004.Active) AND(Ax1.Block) THEN
				ServiceVis.P11.Layers.Layer7 := SHOW ;
			END_IF
		6:
			ServiceVis.P11.Status[6] := SHOW ;
			IF(ServiceLevel.Level > OPERATOR) AND(Tracking10.Busy) THEN
				ServiceVis.P11.Status1[11] := SHOW ;
			END_IF
			IF(Track108.Active) AND(Tracking10.Blocked) THEN
				ServiceVis.P11.Layers.Layer8 := SHOW ;
			END_IF
		7:
			ServiceVis.P11.Status[7] := SHOW ;
			IF(ServiceLevel.Level > OPERATOR) AND(Tracking11.Busy) THEN
				ServiceVis.P11.Status1[12] := SHOW ;
			END_IF
			IF(Track115.Active) AND(Tracking11.Blocked) THEN
				ServiceVis.P11.Layers.Layer9 := SHOW ;
			END_IF
			IF(Track114.Active) AND(Ax2.Block) THEN
				ServiceVis.P11.Layers.Layer10 := SHOW ;
			END_IF
		8:
			ServiceVis.P11.Status[8] := SHOW ;
			IF(Reset.Count) THEN
				Reset.Grind := TRUE ;
				Reset.Time := TRUE ;
			ELSE
				Reset.Grind := FALSE ;
				Reset.Time := FALSE ;
			END_IF
		9:
			ServiceVis.P11.Status[9]	:=	SHOW	;
			IF((Track501.Active) OR(Track601.Active)) AND NOT((Tracking00.Busy) OR(Tracking10.Busy) OR(Tracking11.Busy) OR(Tracking20.Busy) OR(Tracking30.Busy) OR(Tracking30.Busy) OR(Tracking41.Busy) OR(Tracking70.Busy)) THEN //CHANGE TRACKING REGISTER AS REQUIRED
				ServiceVis.P11.Status1[17]	:=	SHOW	;
			END_IF
		10:
			ServiceVis.P11.Status[10]	:=	SHOW	;
		20:
			ServiceVis.P11.Status[20]	:=	SHOW	;
			ServiceVis.Start.Enable	:=	HIDE	;
		21:
			ServiceVis.P11.Status[21]	:=	SHOW	;
		22:
			ServiceVis.P11.Status[22]	:=	SHOW	;
	END_CASE

	IF NOT(Control.Achieved1) THEN
		ServiceVis.P11.Status[16] :=	SHOW	;
	END_IF
	IF NOT(Control.Achieved2) THEN
		ServiceVis.P11.Status[17] :=	SHOW	;
	END_IF
	IF NOT(WashRun.In) THEN
		ServiceVis.P11.Status[18] :=	SHOW	;
	END_IF
	IF NOT(FurnReady.Int) THEN
		ServiceVis.P11.Status[19] :=	SHOW	;
	END_IF

END_PROGRAM
```

### Program Logical/VisControl/ServiceControl/S_Page12 (IEC) - Options screen control

#### S_Page12.st - Cyclic code
```iecst
(********************************************************************
 * COPYRIGHT --
 ********************************************************************
 * Program: S_Page12
 * File: S_Page12.st
 * Author: nicke
 * Created: May 02, 2013
 ********************************************************************
 * Implementation of program S_Page12
 ********************************************************************)

PROGRAM _CYCLIC

	//OPTIONS SCREEN
	ServiceVis.P12.Status[0]	:=	HIDE	;
	ServiceVis.P12.Status[1]	:=	HIDE	;
	ServiceVis.P12.Status[2]	:=	HIDE	;
	ServiceVis.P12.Status[3]	:=	HIDE	;
	ServiceVis.P12.Status[4]	:=	HIDE	;
	ServiceVis.P12.Status[5]	:=	HIDE	;
	ServiceVis.P12.Status[6]	:=	HIDE	;
	ServiceVis.P12.Status[7]	:=	HIDE	;
	ServiceVis.P12.Status[8]	:=	HIDE	;
	ServiceVis.P12.Status[9]	:=	HIDE	;
	ServiceVis.P12.Status[10]	:=	HIDE	;
	ServiceVis.P12.Status[11]	:=	HIDE	;

	CASE ServiceVis.P12.EnableIndex OF
		0:
			ServiceVis.P12.Status[0]	:=	SHOW	;
		1:
			ServiceVis.P12.Status[1]	:=	SHOW	;
		2:
			ServiceVis.P12.Status[2]	:=	SHOW	;
		3:
			ServiceVis.P12.Status[3]	:=	SHOW	;
		4:
			ServiceVis.P12.Status[4]	:=	SHOW	;
		5:
			ServiceVis.P12.Status[5]	:=	SHOW	;
		6:
			ServiceVis.P12.Status[6]	:=	SHOW	;
		7:
			ServiceVis.P12.Status[7]	:=	SHOW	;
		8:
			ServiceVis.P12.Status[8]	:=	SHOW	;
		9:
			ServiceVis.P12.Status[9]	:=	SHOW	;
		10:
			ServiceVis.P12.Status[10]	:=	SHOW	;
	END_CASE
	IF(ServiceLevel.Level > OPERATOR)THEN
		ServiceVis.P12.Status[9]	:=	SHOW	;
	END_IF

	//DISABLE CHANGING BATCHING MODES UNTIL LINE IS EMPTY
	IF(Control.Empty) THEN
		ServiceVis.P12.Status[11]	:=	SHOW	;
	END_IF

	//HIGHLIGHT SELECTED FURNACE CLEAR SIGNAL MODE COLOUR
	CASE LoadPerm.FurnClear OF
		0:
			ServiceVis.P12.Colour[5]	:=	WHITE			;
			ServiceVis.P12.Colour[6]	:=	DROP_UNSELECTED	;
		1:
			ServiceVis.P12.Colour[5]	:=	DROP_UNSELECTED	;
			ServiceVis.P12.Colour[6]	:=	WHITE			;
	END_CASE

END_PROGRAM
```

### Program Logical/VisControl/ServiceControl/S_Page13 (IEC) - Settings screen control
